LIN {X 0,Y 252.245,Z 652.898,A -85,B 0,C 180,E1 -20197.805,E2 -20197.805} C_VEL
LIN {X 0,Y 252.459,Z 653.235,A -85,B 0,C 180,E1 -20199.813,E2 -20199.813} C_VEL
LIN {X 0,Y 253.031,Z 654.37,A -85,B 0,C 180,E1 -20201.806,E2 -20201.806} C_VEL
LIN {X 0,Y 253.295,Z 655.446,A -85,B 0,C 180,E1 -20202.736,E2 -20202.736} C_VEL
LIN {X 0,Y 253.577,Z 657.958,A -85,B 0,C 180,E1 -20203.951,E2 -20203.951} C_VEL
LIN {X 0,Y 253.573,Z 661.43,A -85,B 0,C 180,E1 -20205.049,E2 -20205.049} C_VEL
LIN {X 0,Y 252.747,Z 675.435,A -85,B 0,C 180,E1 -20208.376,E2 -20208.376} C_VEL
LIN {X 0,Y 252.668,Z 684.161,A -85,B 0,C 180,E1 -20210.606,E2 -20210.606} C_VEL
LIN {X 0,Y 251.966,Z 693.895,A -85,B 0,C 180,E1 -20212.79,E2 -20212.79} C_VEL
LIN {X 0,Y 250.461,Z 703.468,A -85,B 0,C 180,E1 -20214.772,E2 -20214.772} C_VEL
LIN {X 0,Y 248.645,Z 710.196,A -85,B 0,C 180,E1 -20216.076,E2 -20216.076} C_VEL
LIN {X 0,Y 244.167,Z 721.841,A -85,B 0,C 180,E1 -20218.314,E2 -20218.314} C_VEL
LIN {X 0,Y 239.831,Z 731.637,A -85,B 0,C 180,E1 -20220.606,E2 -20220.606} C_VEL
LIN {X 0,Y 234.519,Z 741.386,A -85,B 0,C 180,E1 -20223.289,E2 -20223.289} C_VEL
LIN {X 0,Y 230.644,Z 748.224,A -85,B 0,C 180,E1 -20225.712,E2 -20225.712} C_VEL
LIN {X 0,Y 227.208,Z 753.924,A -85,B 0,C 180,E1 -20228.213,E2 -20228.213} C_VEL
LIN {X 0,Y 223.826,Z 759.888,A -85,B 0,C 180,E1 -20231.702,E2 -20231.702} C_VEL
LIN {X 0,Y 221.088,Z 764.261,A -85,B 0,C 180,E1 -20235.269,E2 -20235.269} C_VEL
LIN {X 0,Y 219.589,Z 767.051,A -85,B 0,C 180,E1 -20238.93,E2 -20238.93} C_VEL
LIN {X 0,Y 218.873,Z 768.38,A -85,B 0,C 180,E1 -20242.622,E2 -20242.622} C_VEL
LIN {X 0,Y 218.849,Z 768.456,A -85,B 0,C 180,E1 -20244.579,E2 -20244.579} C_VEL
LIN {X 0,Y 218.925,Z 768.145,A -85,B 0,C 180,E1 -20246.321,E2 -20246.321} C_VEL
LIN {X 0,Y 219.414,Z 766.339,A -85,B 0,C 180,E1 -20250.002,E2 -20250.002} C_VEL
LIN {X 0,Y 219.108,Z 763.745,A -85,B 0,C 180,E1 -20252.759,E2 -20252.759} C_VEL
LIN {X 0,Y 219.216,Z 760.085,A -85,B 0,C 180,E1 -20255.521,E2 -20255.521} C_VEL
LIN {X 0,Y 219.319,Z 755.208,A -85,B 0,C 180,E1 -20258.293,E2 -20258.293} C_VEL
LIN {X 0,Y 219.698,Z 748.98,A -85,B 0,C 180,E1 -20261.067,E2 -20261.067} C_VEL
LIN {X 0,Y 220.582,Z 741.209,A -85,B 0,C 180,E1 -20263.827,E2 -20263.827} C_VEL
LIN {X 0,Y 221.768,Z 731.543,A -85,B 0,C 180,E1 -20266.573,E2 -20266.573} C_VEL
LIN {X 0,Y 223.305,Z 720.643,A -85,B 0,C 180,E1 -20269.027,E2 -20269.027} C_VEL
LIN {X 0,Y 224.735,Z 710.679,A -85,B 0,C 180,E1 -20270.839,E2 -20270.839} C_VEL
LIN {X 0,Y 224.755,Z 697.58,A -85,B 0,C 180,E1 -20272.767,E2 -20272.767} C_VEL
LIN {X 0,Y 224.665,Z 688.245,A -85,B 0,C 180,E1 -20273.997,E2 -20273.997} C_VEL
LIN {X 0,Y 224.567,Z 676.067,A -85,B 0,C 180,E1 -20275.81,E2 -20275.81} C_VEL
LIN {X 0,Y 224.016,Z 662.677,A -85,B 0,C 180,E1 -20277.401,E2 -20277.401} C_VEL
LIN {X 0,Y 222.878,Z 649.109,A -85,B 0,C 180,E1 -20278.629,E2 -20278.629} C_VEL
LIN {X 0,Y 221.828,Z 640.058,A -85,B 0,C 180,E1 -20279.284,E2 -20279.284} C_VEL
LIN {X 0,Y 221.802,Z 634.375,A -85,B 0,C 180,E1 -20280.398,E2 -20280.398} C_VEL
LIN {X 0,Y 223.684,Z 624.514,A -85,B 0,C 180,E1 -20285.785,E2 -20285.785} C_VEL
LIN {X 0,Y 224.829,Z 619.234,A -85,B 0,C 180,E1 -20288.697,E2 -20288.697} C_VEL
LIN {X 0,Y 224.391,Z 614.928,A -85,B 0,C 180,E1 -20291.262,E2 -20291.262} C_VEL
LIN {X 0,Y 222.825,Z 607.241,A -85,B 0,C 180,E1 -20296.06,E2 -20296.06} C_VEL
LIN {X 0,Y 221.557,Z 600.491,A -85,B 0,C 180,E1 -20300.622,E2 -20300.622} C_VEL
LIN {X 0,Y 220.894,Z 596.978,A -85,B 0,C 180,E1 -20303.234,E2 -20303.234} C_VEL
LIN {X 0,Y 220.831,Z 596.982,A -85,B 0,C 180,E1 -20307.245,E2 -20307.245} C_VEL
LIN {X 0,Y 220.842,Z 596.976,A -85,B 0,C 180,E1 -20311.486,E2 -20311.486} C_VEL
LIN {X 0,Y 220.874,Z 596.971,A -85,B 0,C 180,E1 -20315.565,E2 -20315.565} C_VEL
LIN {X 0,Y 220.899,Z 596.97,A -85,B 0,C 180,E1 -20319.514,E2 -20319.514} C_VEL
LIN {X 0,Y 221.023,Z 596.954,A -85,B 0,C 180,E1 -20323.37,E2 -20323.37} C_VEL
LIN {X 0,Y 221.123,Z 596.942,A -85,B 0,C 180,E1 -20329.006,E2 -20329.006} C_VEL
LIN {X 0,Y 221.317,Z 596.917,A -85,B 0,C 180,E1 -20332.702,E2 -20332.702} C_VEL
LIN {X 0,Y 221.517,Z 596.891,A -85,B 0,C 180,E1 -20338.181,E2 -20338.181} C_VEL
LIN {X 0,Y 221.517,Z 596.888,A -85,B 0,C 180,E1 -20341.817,E2 -20341.817} C_VEL
LIN {X 0,Y 221.295,Z 596.913,A -85,B 0,C 180,E1 -20347.297,E2 -20347.297} C_VEL
LIN {X 0,Y 221.117,Z 596.94,A -85,B 0,C 180,E1 -20350.993,E2 -20350.993} C_VEL
LIN {X 0,Y 221.021,Z 596.94,A -85,B 0,C 180,E1 -20356.629,E2 -20356.629} C_VEL
LIN {X 0,Y 220.897,Z 596.97,A -85,B 0,C 180,E1 -20360.485,E2 -20360.485} C_VEL
LIN {X 0,Y 220.871,Z 596.966,A -85,B 0,C 180,E1 -20364.434,E2 -20364.434} C_VEL
LIN {X 0,Y 220.84,Z 596.969,A -85,B 0,C 180,E1 -20368.512,E2 -20368.512} C_VEL
LIN {X 0,Y 220.821,Z 596.977,A -85,B 0,C 180,E1 -20372.755,E2 -20372.755} C_VEL
LIN {X 0,Y 220.813,Z 596.977,A -85,B 0,C 180,E1 -20377.277,E2 -20377.277} C_VEL
LIN {X 0,Y 220.773,Z 596.983,A -85,B 0,C 180,E1 -20381.951,E2 -20381.951} C_VEL
LIN {X 0,Y 220.834,Z 596.974,A -85,B 0,C 180,E1 -20387.051,E2 -20387.051} C_VEL
LIN {X 0,Y 220.813,Z 596.976,A -85,B 0,C 180,E1 -20390.463,E2 -20390.463} C_VEL
LIN {X 0,Y 220.833,Z 596.97,A -85,B 0,C 180,E1 -20392.793,E2 -20392.793} C_VEL
LIN {X 0,Y 220.824,Z 596.973,A -85,B 0,C 180,E1 -20397.244,E2 -20397.244} C_VEL
LIN {X 0,Y 220.828,Z 596.977,A -85,B 0,C 180,E1 -20401.484,E2 -20401.484} C_VEL
LIN {X 0,Y 220.868,Z 596.972,A -85,B 0,C 180,E1 -20405.564,E2 -20405.564} C_VEL
LIN {X 0,Y 220.893,Z 596.969,A -85,B 0,C 180,E1 -20409.512,E2 -20409.512} C_VEL
LIN {X 0,Y 221.017,Z 596.951,A -85,B 0,C 180,E1 -20413.369,E2 -20413.369} C_VEL
LIN {X 0,Y 221.028,Z 596.951,A -85,B 0,C 180,E1 -20416.038,E2 -20416.038} C_VEL
LIN {X 0,Y 223.588,Z 603.871,A -85,B 0,C 180,E1 -20417.009,E2 -20417.009} C_VEL
LIN {X 0,Y 227.422,Z 614.702,A -85,B 0,C 180,E1 -20418.752,E2 -20418.752} C_VEL
LIN {X 0,Y 229.953,Z 624.228,A -85,B 0,C 180,E1 -20420.457,E2 -20420.457} C_VEL
LIN {X 0,Y 230.705,Z 628.301,A -85,B 0,C 180,E1 -20421.237,E2 -20421.237} C_VEL
LIN {X 0,Y 229.152,Z 638.765,A -85,B 0,C 180,E1 -20423.173,E2 -20423.173} C_VEL
LIN {X 0,Y 227.315,Z 649.11,A -85,B 0,C 180,E1 -20425.565,E2 -20425.565} C_VEL
LIN {X 0,Y 225.619,Z 658.089,A -85,B 0,C 180,E1 -20428.213,E2 -20428.213} C_VEL
LIN {X 0,Y 224.289,Z 665.333,A -85,B 0,C 180,E1 -20430.896,E2 -20430.896} C_VEL
LIN {X 0,Y 223.107,Z 671.185,A -85,B 0,C 180,E1 -20433.61,E2 -20433.61} C_VEL
LIN {X 0,Y 222.214,Z 675.812,A -85,B 0,C 180,E1 -20436.354,E2 -20436.354} C_VEL
LIN {X 0,Y 221.701,Z 679.343,A -85,B 0,C 180,E1 -20439.118,E2 -20439.118} C_VEL
LIN {X 0,Y 221.511,Z 681.12,A -85,B 0,C 180,E1 -20440.972,E2 -20440.972} C_VEL
LIN {X 0,Y 221.471,Z 682.492,A -85,B 0,C 180,E1 -20442.833,E2 -20442.833} C_VEL
LIN {X 0,Y 221.569,Z 683.473,A -85,B 0,C 180,E1 -20444.698,E2 -20444.698} C_VEL
LIN {X 0,Y 221.831,Z 684.017,A -85,B 0,C 180,E1 -20446.565,E2 -20446.565} C_VEL
LIN {X 0,Y 222.29,Z 684.143,A -85,B 0,C 180,E1 -20448.473,E2 -20448.473} C_VEL
LIN {X 0,Y 222.808,Z 683.893,A -85,B 0,C 180,E1 -20450.3,E2 -20450.3} C_VEL
LIN {X 0,Y 223.531,Z 683.233,A -85,B 0,C 180,E1 -20452.164,E2 -20452.164} C_VEL
LIN {X 0,Y 225.071,Z 681.267,A -85,B 0,C 180,E1 -20455.105,E2 -20455.105} C_VEL
LIN {X 0,Y 227.381,Z 677.38,A -85,B 0,C 180,E1 -20458.623,E2 -20458.623} C_VEL
LIN {X 0,Y 229.647,Z 673.053,A -85,B 0,C 180,E1 -20461.348,E2 -20461.348} C_VEL
LIN {X 0,Y 232.269,Z 667.442,A -85,B 0,C 180,E1 -20464.038,E2 -20464.038} C_VEL
LIN {X 0,Y 235.317,Z 660.246,A -85,B 0,C 180,E1 -20466.676,E2 -20466.676} C_VEL
LIN {X 0,Y 238.089,Z 652.814,A -85,B 0,C 180,E1 -20468.846,E2 -20468.846} C_VEL
LIN {X 0,Y 239.795,Z 647.581,A -85,B 0,C 180,E1 -20470.147,E2 -20470.147} C_VEL
LIN {X 0,Y 236.234,Z 643.736,A -85,B 0,C 180,E1 -20471.949,E2 -20471.949} C_VEL
LIN {X 0,Y 229.224,Z 637.173,A -85,B 0,C 180,E1 -20475.157,E2 -20475.157} C_VEL
LIN {X 0,Y 223.707,Z 632.758,A -85,B 0,C 180,E1 -20477.512,E2 -20477.512} C_VEL
LIN {X 0,Y 222.648,Z 630.989,A -85,B 0,C 180,E1 -20478.179,E2 -20478.179} C_VEL
LIN {X 0,Y 222.276,Z 635.847,A -85,B 0,C 180,E1 -20480.776,E2 -20480.776} C_VEL
LIN {X 0,Y 224.52,Z 650.074,A -85,B 0,C 180,E1 -20481.923,E2 -20481.923} C_VEL
LIN {X 0,Y 226.528,Z 663.63,A -85,B 0,C 180,E1 -20483.379,E2 -20483.379} C_VEL
LIN {X 0,Y 227.354,Z 670.894,A -85,B 0,C 180,E1 -20484.306,E2 -20484.306} C_VEL
LIN {X 0,Y 225.67,Z 684.053,A -85,B 0,C 180,E1 -20486.175,E2 -20486.175} C_VEL
LIN {X 0,Y 224.013,Z 695.748,A -85,B 0,C 180,E1 -20488.299,E2 -20488.299} C_VEL
LIN {X 0,Y 222.521,Z 706.372,A -85,B 0,C 180,E1 -20490.69,E2 -20490.69} C_VEL
LIN {X 0,Y 221,Z 716.568,A -85,B 0,C 180,E1 -20493.564,E2 -20493.564} C_VEL
LIN {X 0,Y 220.17,Z 723.542,A -85,B 0,C 180,E1 -20495.985,E2 -20495.985} C_VEL
LIN {X 0,Y 219.407,Z 730.071,A -85,B 0,C 180,E1 -20498.772,E2 -20498.772} C_VEL
LIN {X 0,Y 218.933,Z 734.814,A -85,B 0,C 180,E1 -20501.277,E2 -20501.277} C_VEL
LIN {X 0,Y 218.61,Z 739.736,A -85,B 0,C 180,E1 -20504.67,E2 -20504.67} C_VEL
LIN {X 0,Y 218.605,Z 742.265,A -85,B 0,C 180,E1 -20506.995,E2 -20506.995} C_VEL
LIN {X 0,Y 219.038,Z 744.947,A -85,B 0,C 180,E1 -20510.769,E2 -20510.769} C_VEL
LIN {X 0,Y 219.579,Z 745.711,A -85,B 0,C 180,E1 -20512.824,E2 -20512.824} C_VEL
LIN {X 0,Y 220.776,Z 745.89,A -85,B 0,C 180,E1 -20516.35,E2 -20516.35} C_VEL
LIN {X 0,Y 222.836,Z 744.583,A -85,B 0,C 180,E1 -20520.001,E2 -20520.001} C_VEL
LIN {X 0,Y 225.68,Z 741.694,A -85,B 0,C 180,E1 -20523.572,E2 -20523.572} C_VEL
LIN {X 0,Y 228.348,Z 738.462,A -85,B 0,C 180,E1 -20526.185,E2 -20526.185} C_VEL
LIN {X 0,Y 231.512,Z 734.232,A -85,B 0,C 180,E1 -20528.731,E2 -20528.731} C_VEL
LIN {X 0,Y 235.767,Z 727.99,A -85,B 0,C 180,E1 -20531.608,E2 -20531.608} C_VEL
LIN {X 0,Y 240.003,Z 721.133,A -85,B 0,C 180,E1 -20534.004,E2 -20534.004} C_VEL
LIN {X 0,Y 244.573,Z 713.037,A -85,B 0,C 180,E1 -20536.271,E2 -20536.271} C_VEL
LIN {X 0,Y 249.602,Z 703.046,A -85,B 0,C 180,E1 -20538.468,E2 -20538.468} C_VEL
LIN {X 0,Y 252.241,Z 697.161,A -85,B 0,C 180,E1 -20539.533,E2 -20539.533} C_VEL
LIN {X 0,Y 252.802,Z 694.541,A -85,B 0,C 180,E1 -20540.201,E2 -20540.201} C_VEL
LIN {X 0,Y 253.313,Z 686.369,A -85,B 0,C 180,E1 -20542.556,E2 -20542.556} C_VEL
LIN {X 0,Y 253.154,Z 677.893,A -85,B 0,C 180,E1 -20545.251,E2 -20545.251} C_VEL
LIN {X 0,Y 252.633,Z 670.904,A -85,B 0,C 180,E1 -20547.784,E2 -20547.784} C_VEL
LIN {X 0,Y 252.207,Z 668.05,A -85,B 0,C 180,E1 -20549.092,E2 -20549.092} C_VEL
LIN {X 0,Y 251.002,Z 663.368,A -85,B 0,C 180,E1 -20552.141,E2 -20552.141} C_VEL
LIN {X 0,Y 250.022,Z 660.392,A -85,B 0,C 180,E1 -20556.179,E2 -20556.179} C_VEL
LIN {X 0,Y 250.107,Z 659.658,A -85,B 0,C 180,E1 -20558.186,E2 -20558.186} C_VEL
LIN {X 0,Y 250.545,Z 660.411,A -85,B 0,C 180,E1 -20560.77,E2 -20560.77} C_VEL
LIN {X 0,Y 250.953,Z 661.841,A -85,B 0,C 180,E1 -20562.303,E2 -20562.303} C_VEL
LIN {X 0,Y 252.479,Z 667.322,A -85,B 0,C 180,E1 -20565.904,E2 -20565.904} C_VEL
LIN {X 0,Y 252.76,Z 670.488,A -85,B 0,C 180,E1 -20567.023,E2 -20567.023} C_VEL
LIN {X 0,Y 252.747,Z 675.435,A -85,B 0,C 180,E1 -20568.376,E2 -20568.376} C_VEL
LIN {X 0,Y 252.392,Z 679.725,A -85,B 0,C 180,E1 -20569.294,E2 -20569.294} C_VEL
LIN {X 0,Y 251.368,Z 684.518,A -85,B 0,C 180,E1 -20570.061,E2 -20570.061} C_VEL
LIN {X 0,Y 247.481,Z 697.648,A -85,B 0,C 180,E1 -20571.989,E2 -20571.989} C_VEL
LIN {X 0,Y 246.749,Z 700.631,A -85,B 0,C 180,E1 -20572.586,E2 -20572.586} C_VEL
LIN {X 0,Y 244.622,Z 709.219,A -85,B 0,C 180,E1 -20574.429,E2 -20574.429} C_VEL
LIN {X 0,Y 241.616,Z 717.039,A -85,B 0,C 180,E1 -20575.951,E2 -20575.951} C_VEL
LIN {X 0,Y 236.854,Z 727.366,A -85,B 0,C 180,E1 -20578.221,E2 -20578.221} C_VEL
LIN {X 0,Y 232.207,Z 736.247,A -85,B 0,C 180,E1 -20580.542,E2 -20580.542} C_VEL
LIN {X 0,Y 226.841,Z 744.931,A -85,B 0,C 180,E1 -20583.307,E2 -20583.307} C_VEL
LIN {X 0,Y 223.111,Z 751.056,A -85,B 0,C 180,E1 -20585.829,E2 -20585.829} C_VEL
LIN {X 0,Y 219.44,Z 756.501,A -85,B 0,C 180,E1 -20588.648,E2 -20588.648} C_VEL
LIN {X 0,Y 216.301,Z 761.358,A -85,B 0,C 180,E1 -20592.023,E2 -20592.023} C_VEL
LIN {X 0,Y 214.218,Z 764.263,A -85,B 0,C 180,E1 -20594.786,E2 -20594.786} C_VEL
LIN {X 0,Y 212.574,Z 766.842,A -85,B 0,C 180,E1 -20598.56,E2 -20598.56} C_VEL
LIN {X 0,Y 212.1,Z 767.581,A -85,B 0,C 180,E1 -20600.465,E2 -20600.465} C_VEL
LIN {X 0,Y 211.772,Z 767.892,A -85,B 0,C 180,E1 -20604.288,E2 -20604.288} C_VEL
LIN {X 0,Y 211.859,Z 767.493,A -85,B 0,C 180,E1 -20606.198,E2 -20606.198} C_VEL
LIN {X 0,Y 211.921,Z 766.687,A -85,B 0,C 180,E1 -20608.101,E2 -20608.101} C_VEL
LIN {X 0,Y 212.356,Z 765.482,A -85,B 0,C 180,E1 -20610.002,E2 -20610.002} C_VEL
LIN {X 0,Y 212.086,Z 762.722,A -85,B 0,C 180,E1 -20612.851,E2 -20612.851} C_VEL
LIN {X 0,Y 212.159,Z 758.892,A -85,B 0,C 180,E1 -20615.705,E2 -20615.705} C_VEL
LIN {X 0,Y 212.293,Z 753.825,A -85,B 0,C 180,E1 -20618.569,E2 -20618.569} C_VEL
LIN {X 0,Y 212.73,Z 747.381,A -85,B 0,C 180,E1 -20621.435,E2 -20621.435} C_VEL
LIN {X 0,Y 213.635,Z 739.368,A -85,B 0,C 180,E1 -20624.286,E2 -20624.286} C_VEL
LIN {X 0,Y 214.686,Z 731.164,A -85,B 0,C 180,E1 -20626.647,E2 -20626.647} C_VEL
LIN {X 0,Y 216.273,Z 720.163,A -85,B 0,C 180,E1 -20629.205,E2 -20629.205} C_VEL
LIN {X 0,Y 217.672,Z 710.332,A -85,B 0,C 180,E1 -20631.052,E2 -20631.052} C_VEL
LIN {X 0,Y 217.723,Z 699.102,A -85,B 0,C 180,E1 -20632.792,E2 -20632.792} C_VEL
LIN {X 0,Y 217.669,Z 691.704,A -85,B 0,C 180,E1 -20633.805,E2 -20633.805} C_VEL
LIN {X 0,Y 217.728,Z 680.37,A -85,B 0,C 180,E1 -20635.717,E2 -20635.717} C_VEL
LIN {X 0,Y 217.496,Z 667.855,A -85,B 0,C 180,E1 -20637.42,E2 -20637.42} C_VEL
LIN {X 0,Y 216.673,Z 654.932,A -85,B 0,C 180,E1 -20638.808,E2 -20638.808} C_VEL
LIN {X 0,Y 215.186,Z 640.623,A -85,B 0,C 180,E1 -20639.963,E2 -20639.963} C_VEL
LIN {X 0,Y 214.937,Z 638.555,A -85,B 0,C 180,E1 -20640.115,E2 -20640.115} C_VEL
LIN {X 0,Y 214.908,Z 633.563,A -85,B 0,C 180,E1 -20641.14,E2 -20641.14} C_VEL
LIN {X 0,Y 216.56,Z 625.373,A -85,B 0,C 180,E1 -20645.774,E2 -20645.774} C_VEL
LIN {X 0,Y 217.809,Z 619.336,A -85,B 0,C 180,E1 -20649.248,E2 -20649.248} C_VEL
LIN {X 0,Y 217.189,Z 614.995,A -85,B 0,C 180,E1 -20651.904,E2 -20651.904} C_VEL
LIN {X 0,Y 215.661,Z 607.527,A -85,B 0,C 180,E1 -20656.814,E2 -20656.814} C_VEL
LIN {X 0,Y 214.308,Z 600.328,A -85,B 0,C 180,E1 -20661.913,E2 -20661.913} C_VEL
LIN {X 0,Y 213.843,Z 597.857,A -85,B 0,C 180,E1 -20663.839,E2 -20663.839} C_VEL
LIN {X 0,Y 213.802,Z 597.856,A -85,B 0,C 180,E1 -20668.724,E2 -20668.724} C_VEL
LIN {X 0,Y 213.832,Z 597.849,A -85,B 0,C 180,E1 -20672.603,E2 -20672.603} C_VEL
LIN {X 0,Y 213.859,Z 597.845,A -85,B 0,C 180,E1 -20676.953,E2 -20676.953} C_VEL
LIN {X 0,Y 213.95,Z 597.836,A -85,B 0,C 180,E1 -20682.803,E2 -20682.803} C_VEL
LIN {X 0,Y 213.987,Z 597.831,A -85,B 0,C 180,E1 -20686.708,E2 -20686.708} C_VEL
LIN {X 0,Y 214.203,Z 597.804,A -85,B 0,C 180,E1 -20690.557,E2 -20690.557} C_VEL
LIN {X 0,Y 214.254,Z 597.797,A -85,B 0,C 180,E1 -20692.46,E2 -20692.46} C_VEL
LIN {X 0,Y 214.451,Z 597.771,A -85,B 0,C 180,E1 -20698.121,E2 -20698.121} C_VEL
LIN {X 0,Y 214.556,Z 597.759,A -85,B 0,C 180,E1 -20699.999,E2 -20699.999} C_VEL
LIN {X 0,Y 214.45,Z 597.768,A -85,B 0,C 180,E1 -20701.877,E2 -20701.877} C_VEL
LIN {X 0,Y 214.233,Z 597.792,A -85,B 0,C 180,E1 -20707.539,E2 -20707.539} C_VEL
LIN {X 0,Y 214.049,Z 597.82,A -85,B 0,C 180,E1 -20711.361,E2 -20711.361} C_VEL
LIN {X 0,Y 213.936,Z 597.82,A -85,B 0,C 180,E1 -20715.236,E2 -20715.236} C_VEL
LIN {X 0,Y 213.844,Z 597.844,A -85,B 0,C 180,E1 -20719.186,E2 -20719.186} C_VEL
LIN {X 0,Y 213.852,Z 597.843,A -85,B 0,C 180,E1 -20723.226,E2 -20723.226} C_VEL
LIN {X 0,Y 213.833,Z 597.836,A -85,B 0,C 180,E1 -20727.448,E2 -20727.448} C_VEL
LIN {X 0,Y 213.78,Z 597.854,A -85,B 0,C 180,E1 -20731.735,E2 -20731.735} C_VEL
LIN {X 0,Y 213.747,Z 597.86,A -85,B 0,C 180,E1 -20736.287,E2 -20736.287} C_VEL
LIN {X 0,Y 213.715,Z 597.862,A -85,B 0,C 180,E1 -20741.124,E2 -20741.124} C_VEL
LIN {X 0,Y 213.779,Z 597.847,A -85,B 0,C 180,E1 -20746.338,E2 -20746.338} C_VEL
LIN {X 0,Y 213.739,Z 597.852,A -85,B 0,C 180,E1 -20751.335,E2 -20751.335} C_VEL
LIN {X 0,Y 213.771,Z 597.856,A -85,B 0,C 180,E1 -20756.019,E2 -20756.019} C_VEL
LIN {X 0,Y 213.761,Z 597.859,A -85,B 0,C 180,E1 -20760.449,E2 -20760.449} C_VEL
LIN {X 0,Y 213.802,Z 597.853,A -85,B 0,C 180,E1 -20764.7,E2 -20764.7} C_VEL
LIN {X 0,Y 213.814,Z 597.853,A -85,B 0,C 180,E1 -20768.802,E2 -20768.802} C_VEL
LIN {X 0,Y 213.944,Z 597.834,A -85,B 0,C 180,E1 -20772.802,E2 -20772.802} C_VEL
LIN {X 0,Y 213.967,Z 597.91,A -85,B 0,C 180,E1 -20775.233,E2 -20775.233} C_VEL
LIN {X 0,Y 217.501,Z 607.238,A -85,B 0,C 180,E1 -20776.639,E2 -20776.639} C_VEL
LIN {X 0,Y 220.812,Z 616.808,A -85,B 0,C 180,E1 -20778.277,E2 -20778.277} C_VEL
LIN {X 0,Y 223.197,Z 625.637,A -85,B 0,C 180,E1 -20779.944,E2 -20779.944} C_VEL
LIN {X 0,Y 223.95,Z 629.806,A -85,B 0,C 180,E1 -20780.778,E2 -20780.778} C_VEL
LIN {X 0,Y 222.375,Z 640.022,A -85,B 0,C 180,E1 -20782.736,E2 -20782.736} C_VEL
LIN {X 0,Y 220.611,Z 649.483,A -85,B 0,C 180,E1 -20784.972,E2 -20784.972} C_VEL
LIN {X 0,Y 218.837,Z 658.584,A -85,B 0,C 180,E1 -20787.698,E2 -20787.698} C_VEL
LIN {X 0,Y 217.404,Z 665.924,A -85,B 0,C 180,E1 -20790.461,E2 -20790.461} C_VEL
LIN {X 0,Y 215.974,Z 672.721,A -85,B 0,C 180,E1 -20793.73,E2 -20793.73} C_VEL
LIN {X 0,Y 215.119,Z 677.223,A -85,B 0,C 180,E1 -20796.564,E2 -20796.564} C_VEL
LIN {X 0,Y 214.618,Z 680.651,A -85,B 0,C 180,E1 -20799.422,E2 -20799.422} C_VEL
LIN {X 0,Y 214.453,Z 682.376,A -85,B 0,C 180,E1 -20801.338,E2 -20801.338} C_VEL
LIN {X 0,Y 214.441,Z 683.7,A -85,B 0,C 180,E1 -20803.261,E2 -20803.261} C_VEL
LIN {X 0,Y 214.607,Z 684.601,A -85,B 0,C 180,E1 -20805.186,E2 -20805.186} C_VEL
LIN {X 0,Y 215.394,Z 685.157,A -85,B 0,C 180,E1 -20809.042,E2 -20809.042} C_VEL
LIN {X 0,Y 216.007,Z 684.855,A -85,B 0,C 180,E1 -20810.969,E2 -20810.969} C_VEL
LIN {X 0,Y 216.821,Z 684.095,A -85,B 0,C 180,E1 -20812.888,E2 -20812.888} C_VEL
LIN {X 0,Y 218.344,Z 682.239,A -85,B 0,C 180,E1 -20815.678,E2 -20815.678} C_VEL
LIN {X 0,Y 220.274,Z 679.241,A -85,B 0,C 180,E1 -20818.591,E2 -20818.591} C_VEL
LIN {X 0,Y 222.725,Z 674.878,A -85,B 0,C 180,E1 -20821.575,E2 -20821.575} C_VEL
LIN {X 0,Y 225.717,Z 668.854,A -85,B 0,C 180,E1 -20824.625,E2 -20824.625} C_VEL
LIN {X 0,Y 228.61,Z 662.508,A -85,B 0,C 180,E1 -20827.084,E2 -20827.084} C_VEL
LIN {X 0,Y 231.812,Z 654.469,A -85,B 0,C 180,E1 -20829.541,E2 -20829.541} C_VEL
LIN {X 0,Y 233.082,Z 651.055,A -85,B 0,C 180,E1 -20830.428,E2 -20830.428} C_VEL
LIN {X 0,Y 232.462,Z 649.941,A -85,B 0,C 180,E1 -20830.904,E2 -20830.904} C_VEL
LIN {X 0,Y 227.146,Z 644.905,A -85,B 0,C 180,E1 -20833.587,E2 -20833.587} C_VEL
LIN {X 0,Y 222.301,Z 640.532,A -85,B 0,C 180,E1 -20835.932,E2 -20835.932} C_VEL
LIN {X 0,Y 216.034,Z 635.517,A -85,B 0,C 180,E1 -20838.857,E2 -20838.857} C_VEL
LIN {X 0,Y 215.428,Z 634.282,A -85,B 0,C 180,E1 -20839.354,E2 -20839.354} C_VEL
LIN {X 0,Y 215.285,Z 635.964,A -85,B 0,C 180,E1 -20840.29,E2 -20840.29} C_VEL
LIN {X 0,Y 217.629,Z 651.221,A -85,B 0,C 180,E1 -20841.617,E2 -20841.617} C_VEL
LIN {X 0,Y 219.581,Z 664.784,A -85,B 0,C 180,E1 -20843.142,E2 -20843.142} C_VEL
LIN {X 0,Y 220.374,Z 670.376,A -85,B 0,C 180,E1 -20843.887,E2 -20843.887} C_VEL
LIN {X 0,Y 218.947,Z 682,A -85,B 0,C 180,E1 -20845.547,E2 -20845.547} C_VEL
LIN {X 0,Y 217.416,Z 693.05,A -85,B 0,C 180,E1 -20847.5,E2 -20847.5} C_VEL
LIN {X 0,Y 215.939,Z 703.184,A -85,B 0,C 180,E1 -20849.705,E2 -20849.705} C_VEL
LIN {X 0,Y 214.51,Z 712.508,A -85,B 0,C 180,E1 -20852.198,E2 -20852.198} C_VEL
LIN {X 0,Y 213.33,Z 721.502,A -85,B 0,C 180,E1 -20855.164,E2 -20855.164} C_VEL
LIN {X 0,Y 212.527,Z 727.963,A -85,B 0,C 180,E1 -20857.802,E2 -20857.802} C_VEL
LIN {X 0,Y 211.939,Z 733.605,A -85,B 0,C 180,E1 -20860.635,E2 -20860.635} C_VEL
LIN {X 0,Y 211.582,Z 738.416,A -85,B 0,C 180,E1 -20863.7,E2 -20863.7} C_VEL
LIN {X 0,Y 211.485,Z 741.802,A -85,B 0,C 180,E1 -20866.549,E2 -20866.549} C_VEL
LIN {X 0,Y 211.589,Z 743.577,A -85,B 0,C 180,E1 -20868.505,E2 -20868.505} C_VEL
LIN {X 0,Y 211.865,Z 744.921,A -85,B 0,C 180,E1 -20870.454,E2 -20870.454} C_VEL
LIN {X 0,Y 212.485,Z 745.993,A -85,B 0,C 180,E1 -20872.848,E2 -20872.848} C_VEL
LIN {X 0,Y 213.626,Z 746.508,A -85,B 0,C 180,E1 -20876.228,E2 -20876.228} C_VEL
LIN {X 0,Y 215.704,Z 745.599,A -85,B 0,C 180,E1 -20880.001,E2 -20880.001} C_VEL
LIN {X 0,Y 218.617,Z 743.182,A -85,B 0,C 180,E1 -20883.687,E2 -20883.687} C_VEL
LIN {X 0,Y 221.321,Z 740.321,A -85,B 0,C 180,E1 -20886.382,E2 -20886.382} C_VEL
LIN {X 0,Y 224.599,Z 736.503,A -85,B 0,C 180,E1 -20889.002,E2 -20889.002} C_VEL
LIN {X 0,Y 228.331,Z 731.634,A -85,B 0,C 180,E1 -20891.542,E2 -20891.542} C_VEL
LIN {X 0,Y 233.263,Z 724.547,A -85,B 0,C 180,E1 -20894.393,E2 -20894.393} C_VEL
LIN {X 0,Y 238.055,Z 716.965,A -85,B 0,C 180,E1 -20896.73,E2 -20896.73} C_VEL
LIN {X 0,Y 243.241,Z 707.803,A -85,B 0,C 180,E1 -20898.969,E2 -20898.969} C_VEL
LIN {X 0,Y 246.905,Z 700.594,A -85,B 0,C 180,E1 -20900.408,E2 -20900.408} C_VEL
LIN {X 0,Y 247.607,Z 698.809,A -85,B 0,C 180,E1 -20900.782,E2 -20900.782} C_VEL
LIN {X 0,Y 248.563,Z 691.931,A -85,B 0,C 180,E1 -20902.881,E2 -20902.881} C_VEL
LIN {X 0,Y 249,Z 683.501,A -85,B 0,C 180,E1 -20905.703,E2 -20905.703} C_VEL
LIN {X 0,Y 249.005,Z 676.875,A -85,B 0,C 180,E1 -20908.189,E2 -20908.189} C_VEL
LIN {X 0,Y 248.766,Z 673.67,A -85,B 0,C 180,E1 -20909.728,E2 -20909.728} C_VEL
LIN {X 0,Y 248.039,Z 669.604,A -85,B 0,C 180,E1 -20912.572,E2 -20912.572} C_VEL
LIN {X 0,Y 247.521,Z 666.878,A -85,B 0,C 180,E1 -20916.604,E2 -20916.604} C_VEL
LIN {X 0,Y 247.698,Z 666.446,A -85,B 0,C 180,E1 -20918.625,E2 -20918.625} C_VEL
LIN {X 0,Y 248.047,Z 667.091,A -85,B 0,C 180,E1 -20920.668,E2 -20920.668} C_VEL
LIN {X 0,Y 248.449,Z 669.351,A -85,B 0,C 180,E1 -20922.759,E2 -20922.759} C_VEL
LIN {X 0,Y 249.286,Z 672.962,A -85,B 0,C 180,E1 -20925.188,E2 -20925.188} C_VEL
LIN {X 0,Y 249.373,Z 675.951,A -85,B 0,C 180,E1 -20926.295,E2 -20926.295} C_VEL
LIN {X 0,Y 248.73,Z 686.204,A -85,B 0,C 180,E1 -20929.164,E2 -20929.164} C_VEL
LIN {X 0,Y 247.447,Z 696.646,A -85,B 0,C 180,E1 -20931.684,E2 -20931.684} C_VEL
LIN {X 0,Y 246.749,Z 700.631,A -85,B 0,C 180,E1 -20932.586,E2 -20932.586} C_VEL
LIN {X 0,Y 245.893,Z 703.651,A -85,B 0,C 180,E1 -20933.161,E2 -20933.161} C_VEL
LIN {X 0,Y 244.553,Z 706.757,A -85,B 0,C 180,E1 -20933.634,E2 -20933.634} C_VEL
LIN {X 0,Y 240.956,Z 713.132,A -85,B 0,C 180,E1 -20934.405,E2 -20934.405} C_VEL
LIN {X 0,Y 235.938,Z 720.792,A -85,B 0,C 180,E1 -20935.401,E2 -20935.401} C_VEL
LIN {X 0,Y 233.43,Z 725.032,A -85,B 0,C 180,E1 -20936.231,E2 -20936.231} C_VEL
LIN {X 0,Y 227.88,Z 735.142,A -85,B 0,C 180,E1 -20938.899,E2 -20938.899} C_VEL
LIN {X 0,Y 222.133,Z 743.929,A -85,B 0,C 180,E1 -20941.67,E2 -20941.67} C_VEL
LIN {X 0,Y 217.912,Z 750.069,A -85,B 0,C 180,E1 -20944.192,E2 -20944.192} C_VEL
LIN {X 0,Y 213.455,Z 756.156,A -85,B 0,C 180,E1 -20947.405,E2 -20947.405} C_VEL
LIN {X 0,Y 210.378,Z 760.482,A -85,B 0,C 180,E1 -20950.486,E2 -20950.486} C_VEL
LIN {X 0,Y 207.369,Z 764.283,A -85,B 0,C 180,E1 -20954.27,E2 -20954.27} C_VEL
LIN {X 0,Y 205.572,Z 766.581,A -85,B 0,C 180,E1 -20958.165,E2 -20958.165} C_VEL
LIN {X 0,Y 204.771,Z 767.428,A -85,B 0,C 180,E1 -20962.111,E2 -20962.111} C_VEL
LIN {X 0,Y 204.795,Z 766.806,A -85,B 0,C 180,E1 -20966.066,E2 -20966.066} C_VEL
LIN {X 0,Y 205.299,Z 764.571,A -85,B 0,C 180,E1 -20970.002,E2 -20970.002} C_VEL
LIN {X 0,Y 205.063,Z 761.632,A -85,B 0,C 180,E1 -20972.949,E2 -20972.949} C_VEL
LIN {X 0,Y 205.138,Z 757.603,A -85,B 0,C 180,E1 -20975.901,E2 -20975.901} C_VEL
LIN {X 0,Y 205.266,Z 752.318,A -85,B 0,C 180,E1 -20978.865,E2 -20978.865} C_VEL
LIN {X 0,Y 205.768,Z 745.673,A -85,B 0,C 180,E1 -20981.827,E2 -20981.827} C_VEL
LIN {X 0,Y 206.724,Z 737.351,A -85,B 0,C 180,E1 -20984.774,E2 -20984.774} C_VEL
LIN {X 0,Y 207.863,Z 728.899,A -85,B 0,C 180,E1 -20987.21,E2 -20987.21} C_VEL
LIN {X 0,Y 209.384,Z 718.669,A -85,B 0,C 180,E1 -20989.614,E2 -20989.614} C_VEL
LIN {X 0,Y 210.601,Z 709.754,A -85,B 0,C 180,E1 -20991.321,E2 -20991.321} C_VEL
LIN {X 0,Y 210.668,Z 696.957,A -85,B 0,C 180,E1 -20993.34,E2 -20993.34} C_VEL
LIN {X 0,Y 210.68,Z 693.582,A -85,B 0,C 180,E1 -20993.86,E2 -20993.86} C_VEL
LIN {X 0,Y 210.833,Z 681.813,A -85,B 0,C 180,E1 -20996.02,E2 -20996.02} C_VEL
LIN {X 0,Y 210.731,Z 669.4,A -85,B 0,C 180,E1 -20997.835,E2 -20997.835} C_VEL
LIN {X 0,Y 210.08,Z 657.008,A -85,B 0,C 180,E1 -20999.295,E2 -20999.295} C_VEL
LIN {X 0,Y 208.869,Z 643.323,A -85,B 0,C 180,E1 -21000.54,E2 -21000.54} C_VEL
LIN {X 0,Y 208.048,Z 637.114,A -85,B 0,C 180,E1 -21001.01,E2 -21001.01} C_VEL
LIN {X 0,Y 208.053,Z 632.591,A -85,B 0,C 180,E1 -21002.014,E2 -21002.014} C_VEL
LIN {X 0,Y 209.953,Z 624.026,A -85,B 0,C 180,E1 -21007.054,E2 -21007.054} C_VEL
LIN {X 0,Y 210.748,Z 620.203,A -85,B 0,C 180,E1 -21009.319,E2 -21009.319} C_VEL
LIN {X 0,Y 209.954,Z 615.147,A -85,B 0,C 180,E1 -21012.571,E2 -21012.571} C_VEL
LIN {X 0,Y 208.48,Z 607.844,A -85,B 0,C 180,E1 -21017.606,E2 -21017.606} C_VEL
LIN {X 0,Y 207.296,Z 601.32,A -85,B 0,C 180,E1 -21022.391,E2 -21022.391} C_VEL
LIN {X 0,Y 206.77,Z 598.739,A -85,B 0,C 180,E1 -21024.433,E2 -21024.433} C_VEL
LIN {X 0,Y 206.73,Z 598.736,A -85,B 0,C 180,E1 -21029.339,E2 -21029.339} C_VEL
LIN {X 0,Y 206.739,Z 598.732,A -85,B 0,C 180,E1 -21033.772,E2 -21033.772} C_VEL
LIN {X 0,Y 206.765,Z 598.73,A -85,B 0,C 180,E1 -21038.043,E2 -21038.043} C_VEL
LIN {X 0,Y 206.88,Z 598.719,A -85,B 0,C 180,E1 -21042.196,E2 -21042.196} C_VEL
LIN {X 0,Y 206.92,Z 598.715,A -85,B 0,C 180,E1 -21046.245,E2 -21046.245} C_VEL
LIN {X 0,Y 207.139,Z 598.686,A -85,B 0,C 180,E1 -21050.232,E2 -21050.232} C_VEL
LIN {X 0,Y 207.195,Z 598.675,A -85,B 0,C 180,E1 -21052.201,E2 -21052.201} C_VEL
LIN {X 0,Y 207.387,Z 598.651,A -85,B 0,C 180,E1 -21058.057,E2 -21058.057} C_VEL
LIN {X 0,Y 207.521,Z 598.635,A -85,B 0,C 180,E1 -21059.999,E2 -21059.999} C_VEL
LIN {X 0,Y 207.387,Z 598.647,A -85,B 0,C 180,E1 -21061.941,E2 -21061.941} C_VEL
LIN {X 0,Y 207.173,Z 598.672,A -85,B 0,C 180,E1 -21067.798,E2 -21067.798} C_VEL
LIN {X 0,Y 206.986,Z 598.7,A -85,B 0,C 180,E1 -21071.754,E2 -21071.754} C_VEL
LIN {X 0,Y 206.87,Z 598.699,A -85,B 0,C 180,E1 -21075.77,E2 -21075.77} C_VEL
LIN {X 0,Y 206.788,Z 598.723,A -85,B 0,C 180,E1 -21079.868,E2 -21079.868} C_VEL
LIN {X 0,Y 206.768,Z 598.725,A -85,B 0,C 180,E1 -21084.071,E2 -21084.071} C_VEL
LIN {X 0,Y 206.748,Z 598.722,A -85,B 0,C 180,E1 -21088.417,E2 -21088.417} C_VEL
LIN {X 0,Y 206.706,Z 598.734,A -85,B 0,C 180,E1 -21092.955,E2 -21092.955} C_VEL
LIN {X 0,Y 206.683,Z 598.738,A -85,B 0,C 180,E1 -21097.738,E2 -21097.738} C_VEL
LIN {X 0,Y 206.645,Z 598.742,A -85,B 0,C 180,E1 -21101.561,E2 -21101.561} C_VEL
LIN {X 0,Y 206.68,Z 598.728,A -85,B 0,C 180,E1 -21105.567,E2 -21105.567} C_VEL
LIN {X 0,Y 206.681,Z 598.737,A -85,B 0,C 180,E1 -21109.752,E2 -21109.752} C_VEL
LIN {X 0,Y 206.733,Z 598.734,A -85,B 0,C 180,E1 -21114.693,E2 -21114.693} C_VEL
LIN {X 0,Y 206.708,Z 598.734,A -85,B 0,C 180,E1 -21119.335,E2 -21119.335} C_VEL
LIN {X 0,Y 206.733,Z 598.728,A -85,B 0,C 180,E1 -21123.77,E2 -21123.77} C_VEL
LIN {X 0,Y 206.758,Z 598.728,A -85,B 0,C 180,E1 -21128.042,E2 -21128.042} C_VEL
LIN {X 0,Y 206.874,Z 598.718,A -85,B 0,C 180,E1 -21132.195,E2 -21132.195} C_VEL
LIN {X 0,Y 206.882,Z 598.706,A -85,B 0,C 180,E1 -21134.324,E2 -21134.324} C_VEL
LIN {X 0,Y 210.29,Z 607.542,A -85,B 0,C 180,E1 -21135.739,E2 -21135.739} C_VEL
LIN {X 0,Y 214.15,Z 618.59,A -85,B 0,C 180,E1 -21137.716,E2 -21137.716} C_VEL
LIN {X 0,Y 216.696,Z 628.229,A -85,B 0,C 180,E1 -21139.639,E2 -21139.639} C_VEL
LIN {X 0,Y 217.158,Z 630.75,A -85,B 0,C 180,E1 -21140.174,E2 -21140.174} C_VEL
LIN {X 0,Y 215.571,Z 641.287,A -85,B 0,C 180,E1 -21142.27,E2 -21142.27} C_VEL
LIN {X 0,Y 213.909,Z 649.823,A -85,B 0,C 180,E1 -21144.342,E2 -21144.342} C_VEL
LIN {X 0,Y 212.333,Z 657.689,A -85,B 0,C 180,E1 -21146.678,E2 -21146.678} C_VEL
LIN {X 0,Y 210.849,Z 665.053,A -85,B 0,C 180,E1 -21149.377,E2 -21149.377} C_VEL
LIN {X 0,Y 209.632,Z 670.689,A -85,B 0,C 180,E1 -21151.919,E2 -21151.919} C_VEL
LIN {X 0,Y 208.54,Z 675.849,A -85,B 0,C 180,E1 -21154.831,E2 -21154.831} C_VEL
LIN {X 0,Y 207.818,Z 679.872,A -85,B 0,C 180,E1 -21157.772,E2 -21157.772} C_VEL
LIN {X 0,Y 207.463,Z 682.888,A -85,B 0,C 180,E1 -21160.769,E2 -21160.769} C_VEL
LIN {X 0,Y 207.449,Z 684.894,A -85,B 0,C 180,E1 -21163.716,E2 -21163.716} C_VEL
LIN {X 0,Y 208.03,Z 686.13,A -85,B 0,C 180,E1 -21167.699,E2 -21167.699} C_VEL
LIN {X 0,Y 208.544,Z 686.17,A -85,B 0,C 180,E1 -21169.692,E2 -21169.692} C_VEL
LIN {X 0,Y 209.236,Z 685.782,A -85,B 0,C 180,E1 -21171.681,E2 -21171.681} C_VEL
LIN {X 0,Y 210.14,Z 684.956,A -85,B 0,C 180,E1 -21173.659,E2 -21173.659} C_VEL
LIN {X 0,Y 211.631,Z 683.217,A -85,B 0,C 180,E1 -21176.283,E2 -21176.283} C_VEL
LIN {X 0,Y 213.893,Z 679.889,A -85,B 0,C 180,E1 -21179.527,E2 -21179.527} C_VEL
LIN {X 0,Y 216.31,Z 675.797,A -85,B 0,C 180,E1 -21182.356,E2 -21182.356} C_VEL
LIN {X 0,Y 219.208,Z 670.265,A -85,B 0,C 180,E1 -21185.244,E2 -21185.244} C_VEL
LIN {X 0,Y 222.623,Z 663.091,A -85,B 0,C 180,E1 -21188.1,E2 -21188.1} C_VEL
LIN {X 0,Y 226.189,Z 654.487,A -85,B 0,C 180,E1 -21190.728,E2 -21190.728} C_VEL
LIN {X 0,Y 225.355,Z 652.709,A -85,B 0,C 180,E1 -21191.543,E2 -21191.543} C_VEL
LIN {X 0,Y 218.774,Z 646.735,A -85,B 0,C 180,E1 -21195.031,E2 -21195.031} C_VEL
LIN {X 0,Y 210.254,Z 639.917,A -85,B 0,C 180,E1 -21199.323,E2 -21199.323} C_VEL
LIN {X 0,Y 208.838,Z 639.161,A -85,B 0,C 180,E1 -21199.939,E2 -21199.939} C_VEL
LIN {X 0,Y 208.658,Z 638.98,A -85,B 0,C 180,E1 -21200.104,E2 -21200.104} C_VEL
LIN {X 0,Y 210.799,Z 653.071,A -85,B 0,C 180,E1 -21201.386,E2 -21201.386} C_VEL
LIN {X 0,Y 212.566,Z 665.305,A -85,B 0,C 180,E1 -21202.821,E2 -21202.821} C_VEL
LIN {X 0,Y 213.362,Z 671.221,A -85,B 0,C 180,E1 -21203.637,E2 -21203.637} C_VEL
LIN {X 0,Y 211.63,Z 684.377,A -85,B 0,C 180,E1 -21205.63,E2 -21205.63} C_VEL
LIN {X 0,Y 209.888,Z 696.098,A -85,B 0,C 180,E1 -21207.89,E2 -21207.89} C_VEL
LIN {X 0,Y 208.274,Z 707.033,A -85,B 0,C 180,E1 -21210.513,E2 -21210.513} C_VEL
LIN {X 0,Y 206.874,Z 716.2,A -85,B 0,C 180,E1 -21213.249,E2 -21213.249} C_VEL
LIN {X 0,Y 205.842,Z 724.469,A -85,B 0,C 180,E1 -21216.281,E2 -21216.281} C_VEL
LIN {X 0,Y 205.192,Z 730.322,A -85,B 0,C 180,E1 -21218.923,E2 -21218.923} C_VEL
LIN {X 0,Y 204.672,Z 735.813,A -85,B 0,C 180,E1 -21221.999,E2 -21221.999} C_VEL
LIN {X 0,Y 204.433,Z 740.171,A -85,B 0,C 180,E1 -21225.168,E2 -21225.168} C_VEL
LIN {X 0,Y 204.446,Z 743.204,A -85,B 0,C 180,E1 -21228.098,E2 -21228.098} C_VEL
LIN {X 0,Y 205.166,Z 745.903,A -85,B 0,C 180,E1 -21232.125,E2 -21232.125} C_VEL
LIN {X 0,Y 205.744,Z 746.658,A -85,B 0,C 180,E1 -21234.119,E2 -21234.119} C_VEL
LIN {X 0,Y 207.364,Z 746.944,A -85,B 0,C 180,E1 -21238.059,E2 -21238.059} C_VEL
LIN {X 0,Y 209.927,Z 745.737,A -85,B 0,C 180,E1 -21241.919,E2 -21241.919} C_VEL
LIN {X 0,Y 213.298,Z 742.99,A -85,B 0,C 180,E1 -21245.674,E2 -21245.674} C_VEL
LIN {X 0,Y 216.47,Z 739.877,A -85,B 0,C 180,E1 -21248.402,E2 -21248.402} C_VEL
LIN {X 0,Y 221.51,Z 734.242,A -85,B 0,C 180,E1 -21251.902,E2 -21251.902} C_VEL
LIN {X 0,Y 226.575,Z 727.7,A -85,B 0,C 180,E1 -21254.828,E2 -21254.828} C_VEL
LIN {X 0,Y 232.357,Z 719.484,A -85,B 0,C 180,E1 -21257.606,E2 -21257.606} C_VEL
LIN {X 0,Y 237.779,Z 710.743,A -85,B 0,C 180,E1 -21259.872,E2 -21259.872} C_VEL
LIN {X 0,Y 242.341,Z 702.427,A -85,B 0,C 180,E1 -21261.613,E2 -21261.613} C_VEL
LIN {X 0,Y 243.441,Z 698.129,A -85,B 0,C 180,E1 -21262.938,E2 -21262.938} C_VEL
LIN {X 0,Y 244.584,Z 689.689,A -85,B 0,C 180,E1 -21265.892,E2 -21265.892} C_VEL
LIN {X 0,Y 245.205,Z 682.424,A -85,B 0,C 180,E1 -21268.737,E2 -21268.737} C_VEL
LIN {X 0,Y 245.276,Z 680.431,A -85,B 0,C 180,E1 -21269.672,E2 -21269.672} C_VEL
LIN {X 0,Y 244.989,Z 677.076,A -85,B 0,C 180,E1 -21271.924,E2 -21271.924} C_VEL
LIN {X 0,Y 244.868,Z 675.706,A -85,B 0,C 180,E1 -21273.047,E2 -21273.047} C_VEL
LIN {X 0,Y 244.767,Z 673.25,A -85,B 0,C 180,E1 -21277.084,E2 -21277.084} C_VEL
LIN {X 0,Y 245.056,Z 673.146,A -85,B 0,C 180,E1 -21279.258,E2 -21279.258} C_VEL
LIN {X 0,Y 245.376,Z 674.207,A -85,B 0,C 180,E1 -21281.206,E2 -21281.206} C_VEL
LIN {X 0,Y 245.965,Z 678.433,A -85,B 0,C 180,E1 -21284.415,E2 -21284.415} C_VEL
LIN {X 0,Y 245.962,Z 679.797,A -85,B 0,C 180,E1 -21285.034,E2 -21285.034} C_VEL
LIN {X 0,Y 244.898,Z 688.663,A -85,B 0,C 180,E1 -21287.75,E2 -21287.75} C_VEL
LIN {X 0,Y 243.404,Z 697.651,A -85,B 0,C 180,E1 -21290.095,E2 -21290.095} C_VEL
LIN {X 0,Y 241.224,Z 706.76,A -85,B 0,C 180,E1 -21292.28,E2 -21292.28} C_VEL
LIN {X 0,Y 238.607,Z 714.2,A -85,B 0,C 180,E1 -21293.91,E2 -21293.91} C_VEL
LIN {X 0,Y 233.43,Z 725.032,A -85,B 0,C 180,E1 -21296.231,E2 -21296.231} C_VEL
LIN {X 0,Y 230.833,Z 729.13,A -85,B 0,C 180,E1 -21297.093,E2 -21297.093} C_VEL
LIN {X 0,Y 225.038,Z 735.666,A -85,B 0,C 180,E1 -21298.294,E2 -21298.294} C_VEL
LIN {X 0,Y 219.053,Z 741.642,A -85,B 0,C 180,E1 -21299.625,E2 -21299.625} C_VEL
LIN {X 0,Y 216.211,Z 744.853,A -85,B 0,C 180,E1 -21300.685,E2 -21300.685} C_VEL
LIN {X 0,Y 211.607,Z 750.959,A -85,B 0,C 180,E1 -21303.363,E2 -21303.363} C_VEL
LIN {X 0,Y 206.805,Z 756.898,A -85,B 0,C 180,E1 -21306.773,E2 -21306.773} C_VEL
LIN {X 0,Y 203.685,Z 760.778,A -85,B 0,C 180,E1 -21309.818,E2 -21309.818} C_VEL
LIN {X 0,Y 200.543,Z 764.244,A -85,B 0,C 180,E1 -21313.72,E2 -21313.72} C_VEL
LIN {X 0,Y 198.59,Z 766.291,A -85,B 0,C 180,E1 -21317.743,E2 -21317.743} C_VEL
LIN {X 0,Y 197.713,Z 766.922,A -85,B 0,C 180,E1 -21321.828,E2 -21321.828} C_VEL
LIN {X 0,Y 197.733,Z 766.035,A -85,B 0,C 180,E1 -21325.926,E2 -21325.926} C_VEL
LIN {X 0,Y 198.244,Z 763.609,A -85,B 0,C 180,E1 -21330.002,E2 -21330.002} C_VEL
LIN {X 0,Y 198.04,Z 760.509,A -85,B 0,C 180,E1 -21333.053,E2 -21333.053} C_VEL
LIN {X 0,Y 198.097,Z 756.312,A -85,B 0,C 180,E1 -21336.112,E2 -21336.112} C_VEL
LIN {X 0,Y 198.339,Z 749.726,A -85,B 0,C 180,E1 -21339.692,E2 -21339.692} C_VEL
LIN {X 0,Y 198.963,Z 742.537,A -85,B 0,C 180,E1 -21342.756,E2 -21342.756} C_VEL
LIN {X 0,Y 199.869,Z 735.233,A -85,B 0,C 180,E1 -21345.293,E2 -21345.293} C_VEL
LIN {X 0,Y 201.233,Z 725.45,A -85,B 0,C 180,E1 -21348.058,E2 -21348.058} C_VEL
LIN {X 0,Y 202.698,Z 715.727,A -85,B 0,C 180,E1 -21350.289,E2 -21350.289} C_VEL
LIN {X 0,Y 203.534,Z 709.112,A -85,B 0,C 180,E1 -21351.58,E2 -21351.58} C_VEL
LIN {X 0,Y 203.634,Z 695.248,A -85,B 0,C 180,E1 -21353.926,E2 -21353.926} C_VEL
LIN {X 0,Y 203.925,Z 684.613,A -85,B 0,C 180,E1 -21356.061,E2 -21356.061} C_VEL
LIN {X 0,Y 203.989,Z 672.779,A -85,B 0,C 180,E1 -21357.998,E2 -21357.998} C_VEL
LIN {X 0,Y 203.594,Z 660.701,A -85,B 0,C 180,E1 -21359.604,E2 -21359.604} C_VEL
LIN {X 0,Y 202.624,Z 647.447,A -85,B 0,C 180,E1 -21360.992,E2 -21360.992} C_VEL
LIN {X 0,Y 201.153,Z 635.493,A -85,B 0,C 180,E1 -21361.968,E2 -21361.968} C_VEL
LIN {X 0,Y 201.222,Z 631.683,A -85,B 0,C 180,E1 -21362.895,E2 -21362.895} C_VEL
LIN {X 0,Y 203.413,Z 622.59,A -85,B 0,C 180,E1 -21368.457,E2 -21368.457} C_VEL
LIN {X 0,Y 203.7,Z 620.988,A -85,B 0,C 180,E1 -21369.445,E2 -21369.445} C_VEL
LIN {X 0,Y 203.092,Z 616.904,A -85,B 0,C 180,E1 -21372.17,E2 -21372.17} C_VEL
LIN {X 0,Y 201.658,Z 609.964,A -85,B 0,C 180,E1 -21377.046,E2 -21377.046} C_VEL
LIN {X 0,Y 200.433,Z 603.218,A -85,B 0,C 180,E1 -21382.147,E2 -21382.147} C_VEL
LIN {X 0,Y 199.726,Z 599.616,A -85,B 0,C 180,E1 -21385.045,E2 -21385.045} C_VEL
LIN {X 0,Y 199.711,Z 599.614,A -85,B 0,C 180,E1 -21388.138,E2 -21388.138} C_VEL
LIN {X 0,Y 199.693,Z 599.61,A -85,B 0,C 180,E1 -21392.772,E2 -21392.772} C_VEL
LIN {X 0,Y 199.745,Z 599.603,A -85,B 0,C 180,E1 -21397.229,E2 -21397.229} C_VEL
LIN {X 0,Y 199.803,Z 599.599,A -85,B 0,C 180,E1 -21401.757,E2 -21401.757} C_VEL
LIN {X 0,Y 199.854,Z 599.593,A -85,B 0,C 180,E1 -21405.749,E2 -21405.749} C_VEL
LIN {X 0,Y 200.082,Z 599.564,A -85,B 0,C 180,E1 -21409.884,E2 -21409.884} C_VEL
LIN {X 0,Y 200.138,Z 599.554,A -85,B 0,C 180,E1 -21411.925,E2 -21411.925} C_VEL
LIN {X 0,Y 200.327,Z 599.53,A -85,B 0,C 180,E1 -21417.989,E2 -21417.989} C_VEL
LIN {X 0,Y 200.485,Z 599.512,A -85,B 0,C 180,E1 -21419.999,E2 -21419.999} C_VEL
LIN {X 0,Y 200.034,Z 599.551,A -85,B 0,C 180,E1 -21424.029,E2 -21424.029} C_VEL
LIN {X 0,Y 200.117,Z 599.552,A -85,B 0,C 180,E1 -21428.075,E2 -21428.075} C_VEL
LIN {X 0,Y 199.918,Z 599.581,A -85,B 0,C 180,E1 -21432.176,E2 -21432.176} C_VEL
LIN {X 0,Y 199.808,Z 599.578,A -85,B 0,C 180,E1 -21436.342,E2 -21436.342} C_VEL
LIN {X 0,Y 199.705,Z 599.61,A -85,B 0,C 180,E1 -21440.604,E2 -21440.604} C_VEL
LIN {X 0,Y 199.677,Z 599.602,A -85,B 0,C 180,E1 -21444.983,E2 -21444.983} C_VEL
LIN {X 0,Y 199.679,Z 599.607,A -85,B 0,C 180,E1 -21449.521,E2 -21449.521} C_VEL
LIN {X 0,Y 199.681,Z 599.613,A -85,B 0,C 180,E1 -21452.357,E2 -21452.357} C_VEL
LIN {X 0,Y 199.626,Z 599.618,A -85,B 0,C 180,E1 -21456.761,E2 -21456.761} C_VEL
LIN {X 0,Y 199.611,Z 599.617,A -85,B 0,C 180,E1 -21459.326,E2 -21459.326} C_VEL
LIN {X 0,Y 199.578,Z 599.622,A -85,B 0,C 180,E1 -21462.309,E2 -21462.309} C_VEL
LIN {X 0,Y 199.614,Z 599.607,A -85,B 0,C 180,E1 -21465.236,E2 -21465.236} C_VEL
LIN {X 0,Y 199.624,Z 599.616,A -85,B 0,C 180,E1 -21468.014,E2 -21468.014} C_VEL
LIN {X 0,Y 199.644,Z 599.609,A -85,B 0,C 180,E1 -21470.754,E2 -21470.754} C_VEL
LIN {X 0,Y 199.635,Z 599.616,A -85,B 0,C 180,E1 -21475.716,E2 -21475.716} C_VEL
LIN {X 0,Y 199.698,Z 599.603,A -85,B 0,C 180,E1 -21478.135,E2 -21478.135} C_VEL
LIN {X 0,Y 199.686,Z 599.606,A -85,B 0,C 180,E1 -21482.77,E2 -21482.77} C_VEL
LIN {X 0,Y 199.739,Z 599.601,A -85,B 0,C 180,E1 -21487.227,E2 -21487.227} C_VEL
LIN {X 0,Y 199.813,Z 599.594,A -85,B 0,C 180,E1 -21492.709,E2 -21492.709} C_VEL
LIN {X 0,Y 199.826,Z 599.733,A -85,B 0,C 180,E1 -21493.42,E2 -21493.42} C_VEL
LIN {X 0,Y 201.719,Z 604.613,A -85,B 0,C 180,E1 -21494.205,E2 -21494.205} C_VEL
LIN {X 0,Y 205.902,Z 615.529,A -85,B 0,C 180,E1 -21496.175,E2 -21496.175} C_VEL
LIN {X 0,Y 208.807,Z 624.97,A -85,B 0,C 180,E1 -21498.063,E2 -21498.063} C_VEL
LIN {X 0,Y 210.456,Z 632.692,A -85,B 0,C 180,E1 -21499.743,E2 -21499.743} C_VEL
LIN {X 0,Y 208.588,Z 643.598,A -85,B 0,C 180,E1 -21502.009,E2 -21502.009} C_VEL
LIN {X 0,Y 206.565,Z 653.522,A -85,B 0,C 180,E1 -21504.63,E2 -21504.63} C_VEL
LIN {X 0,Y 204.74,Z 662.266,A -85,B 0,C 180,E1 -21507.539,E2 -21507.539} C_VEL
LIN {X 0,Y 203.229,Z 669.283,A -85,B 0,C 180,E1 -21510.494,E2 -21510.494} C_VEL
LIN {X 0,Y 201.761,Z 675.756,A -85,B 0,C 180,E1 -21513.993,E2 -21513.993} C_VEL
LIN {X 0,Y 200.921,Z 680.039,A -85,B 0,C 180,E1 -21517.03,E2 -21517.03} C_VEL
LIN {X 0,Y 200.471,Z 683.26,A -85,B 0,C 180,E1 -21520.093,E2 -21520.093} C_VEL
LIN {X 0,Y 200.37,Z 684.885,A -85,B 0,C 180,E1 -21522.147,E2 -21522.147} C_VEL
LIN {X 0,Y 200.442,Z 686.054,A -85,B 0,C 180,E1 -21524.206,E2 -21524.206} C_VEL
LIN {X 0,Y 201.139,Z 687.191,A -85,B 0,C 180,E1 -21528.327,E2 -21528.327} C_VEL
LIN {X 0,Y 201.736,Z 687.165,A -85,B 0,C 180,E1 -21530.386,E2 -21530.386} C_VEL
LIN {X 0,Y 202.493,Z 686.695,A -85,B 0,C 180,E1 -21532.442,E2 -21532.442} C_VEL
LIN {X 0,Y 203.514,Z 685.816,A -85,B 0,C 180,E1 -21534.479,E2 -21534.479} C_VEL
LIN {X 0,Y 204.929,Z 684.208,A -85,B 0,C 180,E1 -21536.919,E2 -21536.919} C_VEL
LIN {X 0,Y 207.561,Z 680.544,A -85,B 0,C 180,E1 -21540.522,E2 -21540.522} C_VEL
LIN {X 0,Y 210.31,Z 676.1,A -85,B 0,C 180,E1 -21543.569,E2 -21543.569} C_VEL
LIN {X 0,Y 213.285,Z 670.681,A -85,B 0,C 180,E1 -21546.376,E2 -21546.376} C_VEL
LIN {X 0,Y 216.721,Z 663.665,A -85,B 0,C 180,E1 -21549.169,E2 -21549.169} C_VEL
LIN {X 0,Y 219.296,Z 657.925,A -85,B 0,C 180,E1 -21551.012,E2 -21551.012} C_VEL
LIN {X 0,Y 219.335,Z 656.604,A -85,B 0,C 180,E1 -21551.507,E2 -21551.507} C_VEL
LIN {X 0,Y 213.356,Z 651.321,A -85,B 0,C 180,E1 -21554.911,E2 -21554.911} C_VEL
LIN {X 0,Y 207.072,Z 646.346,A -85,B 0,C 180,E1 -21558.3,E2 -21558.3} C_VEL
LIN {X 0,Y 204.469,Z 645.902,A -85,B 0,C 180,E1 -21559.228,E2 -21559.228} C_VEL
LIN {X 0,Y 202.544,Z 644.928,A -85,B 0,C 180,E1 -21560.138,E2 -21560.138} C_VEL
LIN {X 0,Y 204.836,Z 660.756,A -85,B 0,C 180,E1 -21561.861,E2 -21561.861} C_VEL
LIN {X 0,Y 206.294,Z 671.973,A -85,B 0,C 180,E1 -21563.404,E2 -21563.404} C_VEL
LIN {X 0,Y 204.715,Z 683.536,A -85,B 0,C 180,E1 -21565.199,E2 -21565.199} C_VEL
LIN {X 0,Y 202.922,Z 695.536,A -85,B 0,C 180,E1 -21567.533,E2 -21567.533} C_VEL
LIN {X 0,Y 201.307,Z 706.34,A -85,B 0,C 180,E1 -21570.167,E2 -21570.167} C_VEL
LIN {X 0,Y 199.93,Z 715.197,A -85,B 0,C 180,E1 -21572.808,E2 -21572.808} C_VEL
LIN {X 0,Y 198.808,Z 723.831,A -85,B 0,C 180,E1 -21576.015,E2 -21576.015} C_VEL
LIN {X 0,Y 198.042,Z 730.759,A -85,B 0,C 180,E1 -21579.215,E2 -21579.215} C_VEL
LIN {X 0,Y 197.546,Z 736.236,A -85,B 0,C 180,E1 -21582.399,E2 -21582.399} C_VEL
LIN {X 0,Y 197.314,Z 740.481,A -85,B 0,C 180,E1 -21585.563,E2 -21585.563} C_VEL
LIN {X 0,Y 197.317,Z 742.694,A -85,B 0,C 180,E1 -21587.661,E2 -21587.661} C_VEL
LIN {X 0,Y 197.564,Z 744.482,A -85,B 0,C 180,E1 -21589.755,E2 -21589.755} C_VEL
LIN {X 0,Y 198.289,Z 746.381,A -85,B 0,C 180,E1 -21592.917,E2 -21592.917} C_VEL
LIN {X 0,Y 199.276,Z 747.352,A -85,B 0,C 180,E1 -21595.956,E2 -21595.956} C_VEL
LIN {X 0,Y 201.388,Z 747.357,A -85,B 0,C 180,E1 -21600.001,E2 -21600.001} C_VEL
LIN {X 0,Y 204.416,Z 745.812,A -85,B 0,C 180,E1 -21603.944,E2 -21603.944} C_VEL
LIN {X 0,Y 208.364,Z 742.787,A -85,B 0,C 180,E1 -21607.755,E2 -21607.755} C_VEL
LIN {X 0,Y 211.986,Z 739.456,A -85,B 0,C 180,E1 -21610.507,E2 -21610.507} C_VEL
LIN {X 0,Y 217.014,Z 734.064,A -85,B 0,C 180,E1 -21613.709,E2 -21613.709} C_VEL
LIN {X 0,Y 222.354,Z 727.709,A -85,B 0,C 180,E1 -21616.528,E2 -21616.528} C_VEL
LIN {X 0,Y 227.633,Z 720.688,A -85,B 0,C 180,E1 -21618.917,E2 -21618.917} C_VEL
LIN {X 0,Y 233.351,Z 712.168,A -85,B 0,C 180,E1 -21621.188,E2 -21621.188} C_VEL
LIN {X 0,Y 237.369,Z 705.543,A -85,B 0,C 180,E1 -21622.638,E2 -21622.638} C_VEL
LIN {X 0,Y 238.338,Z 702.797,A -85,B 0,C 180,E1 -21623.46,E2 -21623.46} C_VEL
LIN {X 0,Y 239.901,Z 695.715,A -85,B 0,C 180,E1 -21626.068,E2 -21626.068} C_VEL
LIN {X 0,Y 241.174,Z 688.372,A -85,B 0,C 180,E1 -21629.051,E2 -21629.051} C_VEL
LIN {X 0,Y 241.494,Z 685.185,A -85,B 0,C 180,E1 -21630.718,E2 -21630.718} C_VEL
LIN {X 0,Y 241.475,Z 682.867,A -85,B 0,C 180,E1 -21632.436,E2 -21632.436} C_VEL
LIN {X 0,Y 241.509,Z 681.716,A -85,B 0,C 180,E1 -21633.567,E2 -21633.567} C_VEL
LIN {X 0,Y 241.416,Z 680.42,A -85,B 0,C 180,E1 -21635.608,E2 -21635.608} C_VEL
LIN {X 0,Y 241.794,Z 679.555,A -85,B 0,C 180,E1 -21638.302,E2 -21638.302} C_VEL
LIN {X 0,Y 242.044,Z 679.809,A -85,B 0,C 180,E1 -21639.703,E2 -21639.703} C_VEL
LIN {X 0,Y 242.226,Z 680.594,A -85,B 0,C 180,E1 -21641.033,E2 -21641.033} C_VEL
LIN {X 0,Y 242.419,Z 683.726,A -85,B 0,C 180,E1 -21643.552,E2 -21643.552} C_VEL
LIN {X 0,Y 242.456,Z 684.651,A -85,B 0,C 180,E1 -21644.082,E2 -21644.082} C_VEL
LIN {X 0,Y 241.705,Z 688.71,A -85,B 0,C 180,E1 -21645.498,E2 -21645.498} C_VEL
LIN {X 0,Y 240.209,Z 696.123,A -85,B 0,C 180,E1 -21647.709,E2 -21647.709} C_VEL
LIN {X 0,Y 237.738,Z 705.612,A -85,B 0,C 180,E1 -21650.23,E2 -21650.23} C_VEL
LIN {X 0,Y 235.122,Z 713.058,A -85,B 0,C 180,E1 -21652.043,E2 -21652.043} C_VEL
LIN {X 0,Y 231.511,Z 720.677,A -85,B 0,C 180,E1 -21653.706,E2 -21653.706} C_VEL
LIN {X 0,Y 225.364,Z 731.488,A -85,B 0,C 180,E1 -21656.392,E2 -21656.392} C_VEL
LIN {X 0,Y 220.214,Z 739.443,A -85,B 0,C 180,E1 -21658.763,E2 -21658.763} C_VEL
LIN {X 0,Y 216.211,Z 744.853,A -85,B 0,C 180,E1 -21660.685,E2 -21660.685} C_VEL
LIN {X 0,Y 213.385,Z 747.94,A -85,B 0,C 180,E1 -21661.819,E2 -21661.819} C_VEL
LIN {X 0,Y 207.381,Z 752.632,A -85,B 0,C 180,E1 -21663.568,E2 -21663.568} C_VEL
LIN {X 0,Y 201.622,Z 756.621,A -85,B 0,C 180,E1 -21665.51,E2 -21665.51} C_VEL
LIN {X 0,Y 199.232,Z 758.607,A -85,B 0,C 180,E1 -21666.922,E2 -21666.922} C_VEL
LIN {X 0,Y 195.272,Z 762.767,A -85,B 0,C 180,E1 -21671.102,E2 -21671.102} C_VEL
LIN {X 0,Y 192.466,Z 765.272,A -85,B 0,C 180,E1 -21675.192,E2 -21675.192} C_VEL
LIN {X 0,Y 191.029,Z 766.329,A -85,B 0,C 180,E1 -21679.402,E2 -21679.402} C_VEL
LIN {X 0,Y 190.575,Z 765.963,A -85,B 0,C 180,E1 -21683.65,E2 -21683.65} C_VEL
LIN {X 0,Y 190.672,Z 765.247,A -85,B 0,C 180,E1 -21685.774,E2 -21685.774} C_VEL
LIN {X 0,Y 190.802,Z 764.131,A -85,B 0,C 180,E1 -21687.891,E2 -21687.891} C_VEL
LIN {X 0,Y 191.208,Z 762.576,A -85,B 0,C 180,E1 -21690.002,E2 -21690.002} C_VEL
LIN {X 0,Y 191.018,Z 759.28,A -85,B 0,C 180,E1 -21693.166,E2 -21693.166} C_VEL
LIN {X 0,Y 191.108,Z 754.079,A -85,B 0,C 180,E1 -21696.813,E2 -21696.813} C_VEL
LIN {X 0,Y 191.37,Z 748.059,A -85,B 0,C 180,E1 -21700.048,E2 -21700.048} C_VEL
LIN {X 0,Y 192.06,Z 740.617,A -85,B 0,C 180,E1 -21703.223,E2 -21703.223} C_VEL
LIN {X 0,Y 193.286,Z 731.338,A -85,B 0,C 180,E1 -21706.369,E2 -21706.369} C_VEL
LIN {X 0,Y 194.831,Z 720.757,A -85,B 0,C 180,E1 -21709.22,E2 -21709.22} C_VEL
LIN {X 0,Y 196.457,Z 709.981,A -85,B 0,C 180,E1 -21711.545,E2 -21711.545} C_VEL
LIN {X 0,Y 196.563,Z 697.914,A -85,B 0,C 180,E1 -21713.72,E2 -21713.72} C_VEL
LIN {X 0,Y 197.006,Z 686.717,A -85,B 0,C 180,E1 -21716.196,E2 -21716.196} C_VEL
LIN {X 0,Y 197.201,Z 675.787,A -85,B 0,C 180,E1 -21718.18,E2 -21718.18} C_VEL
LIN {X 0,Y 197.017,Z 663.755,A -85,B 0,C 180,E1 -21719.963,E2 -21719.963} C_VEL
LIN {X 0,Y 196.192,Z 649.963,A -85,B 0,C 180,E1 -21721.57,E2 -21721.57} C_VEL
LIN {X 0,Y 194.746,Z 636.882,A -85,B 0,C 180,E1 -21722.755,E2 -21722.755} C_VEL
LIN {X 0,Y 194.299,Z 633.772,A -85,B 0,C 180,E1 -21723.03,E2 -21723.03} C_VEL
LIN {X 0,Y 194.412,Z 630.951,A -85,B 0,C 180,E1 -21723.75,E2 -21723.75} C_VEL
LIN {X 0,Y 196.434,Z 622.882,A -85,B 0,C 180,E1 -21728.873,E2 -21728.873} C_VEL
LIN {X 0,Y 196.58,Z 621.07,A -85,B 0,C 180,E1 -21730.057,E2 -21730.057} C_VEL
LIN {X 0,Y 195.546,Z 615.378,A -85,B 0,C 180,E1 -21734.043,E2 -21734.043} C_VEL
LIN {X 0,Y 194.115,Z 608.134,A -85,B 0,C 180,E1 -21739.494,E2 -21739.494} C_VEL
LIN {X 0,Y 192.979,Z 602.102,A -85,B 0,C 180,E1 -21744.359,E2 -21744.359} C_VEL
LIN {X 0,Y 192.625,Z 600.5,A -85,B 0,C 180,E1 -21745.877,E2 -21745.877} C_VEL
LIN {X 0,Y 192.657,Z 600.487,A -85,B 0,C 180,E1 -21751.108,E2 -21751.108} C_VEL
LIN {X 0,Y 192.713,Z 600.482,A -85,B 0,C 180,E1 -21756.349,E2 -21756.349} C_VEL
LIN {X 0,Y 192.739,Z 600.478,A -85,B 0,C 180,E1 -21761.457,E2 -21761.457} C_VEL
LIN {X 0,Y 192.778,Z 600.474,A -85,B 0,C 180,E1 -21765.214,E2 -21765.214} C_VEL
LIN {X 0,Y 193.027,Z 600.442,A -85,B 0,C 180,E1 -21769.51,E2 -21769.51} C_VEL
LIN {X 0,Y 193.01,Z 600.442,A -85,B 0,C 180,E1 -21773.728,E2 -21773.728} C_VEL
LIN {X 0,Y 193.269,Z 600.409,A -85,B 0,C 180,E1 -21777.915,E2 -21777.915} C_VEL
LIN {X 0,Y 193.449,Z 600.388,A -85,B 0,C 180,E1 -21779.999,E2 -21779.999} C_VEL
LIN {X 0,Y 192.98,Z 600.427,A -85,B 0,C 180,E1 -21784.176,E2 -21784.176} C_VEL
LIN {X 0,Y 193.068,Z 600.432,A -85,B 0,C 180,E1 -21788.372,E2 -21788.372} C_VEL
LIN {X 0,Y 192.857,Z 600.457,A -85,B 0,C 180,E1 -21792.629,E2 -21792.629} C_VEL
LIN {X 0,Y 192.762,Z 600.458,A -85,B 0,C 180,E1 -21796.957,E2 -21796.957} C_VEL
LIN {X 0,Y 192.641,Z 600.487,A -85,B 0,C 180,E1 -21801.396,E2 -21801.396} C_VEL
LIN {X 0,Y 192.669,Z 600.479,A -85,B 0,C 180,E1 -21804.223,E2 -21804.223} C_VEL
LIN {X 0,Y 192.654,Z 600.481,A -85,B 0,C 180,E1 -21808.891,E2 -21808.891} C_VEL
LIN {X 0,Y 192.602,Z 600.49,A -85,B 0,C 180,E1 -21813.184,E2 -21813.184} C_VEL
LIN {X 0,Y 192.554,Z 600.497,A -85,B 0,C 180,E1 -21818.35,E2 -21818.35} C_VEL
LIN {X 0,Y 192.519,Z 600.497,A -85,B 0,C 180,E1 -21823.102,E2 -21823.102} C_VEL
LIN {X 0,Y 192.549,Z 600.495,A -85,B 0,C 180,E1 -21826.885,E2 -21826.885} C_VEL
LIN {X 0,Y 192.577,Z 600.487,A -85,B 0,C 180,E1 -21831.652,E2 -21831.652} C_VEL
LIN {X 0,Y 192.6,Z 600.491,A -85,B 0,C 180,E1 -21834.277,E2 -21834.277} C_VEL
LIN {X 0,Y 192.601,Z 600.49,A -85,B 0,C 180,E1 -21839.277,E2 -21839.277} C_VEL
LIN {X 0,Y 192.662,Z 600.486,A -85,B 0,C 180,E1 -21841.689,E2 -21841.689} C_VEL
LIN {X 0,Y 192.707,Z 600.479,A -85,B 0,C 180,E1 -21846.347,E2 -21846.347} C_VEL
LIN {X 0,Y 192.79,Z 600.608,A -85,B 0,C 180,E1 -21852.406,E2 -21852.406} C_VEL
LIN {X 0,Y 195.065,Z 606.32,A -85,B 0,C 180,E1 -21853.384,E2 -21853.384} C_VEL
LIN {X 0,Y 199.097,Z 616.909,A -85,B 0,C 180,E1 -21855.406,E2 -21855.406} C_VEL
LIN {X 0,Y 202.131,Z 626.683,A -85,B 0,C 180,E1 -21857.471,E2 -21857.471} C_VEL
LIN {X 0,Y 203.587,Z 632.873,A -85,B 0,C 180,E1 -21858.894,E2 -21858.894} C_VEL
LIN {X 0,Y 203.687,Z 634.68,A -85,B 0,C 180,E1 -21859.288,E2 -21859.288} C_VEL
LIN {X 0,Y 201.822,Z 644.821,A -85,B 0,C 180,E1 -21861.487,E2 -21861.487} C_VEL
LIN {X 0,Y 199.882,Z 653.902,A -85,B 0,C 180,E1 -21863.943,E2 -21863.943} C_VEL
LIN {X 0,Y 197.962,Z 662.749,A -85,B 0,C 180,E1 -21866.946,E2 -21866.946} C_VEL
LIN {X 0,Y 196.376,Z 669.892,A -85,B 0,C 180,E1 -21869.998,E2 -21869.998} C_VEL
LIN {X 0,Y 195.013,Z 675.629,A -85,B 0,C 180,E1 -21873.097,E2 -21873.097} C_VEL
LIN {X 0,Y 194.044,Z 680.168,A -85,B 0,C 180,E1 -21876.236,E2 -21876.236} C_VEL
LIN {X 0,Y 193.663,Z 682.572,A -85,B 0,C 180,E1 -21878.344,E2 -21878.344} C_VEL
LIN {X 0,Y 193.368,Z 685.056,A -85,B 0,C 180,E1 -21881.097,E2 -21881.097} C_VEL
LIN {X 0,Y 193.474,Z 687.205,A -85,B 0,C 180,E1 -21884.729,E2 -21884.729} C_VEL
LIN {X 0,Y 194.265,Z 688.25,A -85,B 0,C 180,E1 -21889,E2 -21889} C_VEL
LIN {X 0,Y 194.947,Z 688.129,A -85,B 0,C 180,E1 -21891.129,E2 -21891.129} C_VEL
LIN {X 0,Y 195.809,Z 687.607,A -85,B 0,C 180,E1 -21893.252,E2 -21893.252} C_VEL
LIN {X 0,Y 196.902,Z 686.684,A -85,B 0,C 180,E1 -21895.358,E2 -21895.358} C_VEL
LIN {X 0,Y 198.267,Z 685.193,A -85,B 0,C 180,E1 -21897.605,E2 -21897.605} C_VEL
LIN {X 0,Y 200.444,Z 682.413,A -85,B 0,C 180,E1 -21900.555,E2 -21900.555} C_VEL
LIN {X 0,Y 203.619,Z 677.649,A -85,B 0,C 180,E1 -21904.07,E2 -21904.07} C_VEL
LIN {X 0,Y 206.846,Z 672.103,A -85,B 0,C 180,E1 -21907.089,E2 -21907.089} C_VEL
LIN {X 0,Y 210.432,Z 665.245,A -85,B 0,C 180,E1 -21909.944,E2 -21909.944} C_VEL
LIN {X 0,Y 212.491,Z 660.907,A -85,B 0,C 180,E1 -21911.411,E2 -21911.411} C_VEL
LIN {X 0,Y 211.895,Z 659.266,A -85,B 0,C 180,E1 -21912.263,E2 -21912.263} C_VEL
LIN {X 0,Y 207.827,Z 655.745,A -85,B 0,C 180,E1 -21914.754,E2 -21914.754} C_VEL
LIN {X 0,Y 204.557,Z 653.345,A -85,B 0,C 180,E1 -21916.597,E2 -21916.597} C_VEL
LIN {X 0,Y 201.023,Z 651.377,A -85,B 0,C 180,E1 -21918.375,E2 -21918.375} C_VEL
LIN {X 0,Y 196.614,Z 650.986,A -85,B 0,C 180,E1 -21919.954,E2 -21919.954} C_VEL
LIN {X 0,Y 196.252,Z 650.536,A -85,B 0,C 180,E1 -21920.242,E2 -21920.242} C_VEL
LIN {X 0,Y 198.236,Z 664.5,A -85,B 0,C 180,E1 -21921.948,E2 -21921.948} C_VEL
LIN {X 0,Y 199.227,Z 672.721,A -85,B 0,C 180,E1 -21923.153,E2 -21923.153} C_VEL
LIN {X 0,Y 197.385,Z 685.697,A -85,B 0,C 180,E1 -21925.272,E2 -21925.272} C_VEL
LIN {X 0,Y 195.643,Z 697.308,A -85,B 0,C 180,E1 -21927.701,E2 -21927.701} C_VEL
LIN {X 0,Y 194.032,Z 707.62,A -85,B 0,C 180,E1 -21930.373,E2 -21930.373} C_VEL
LIN {X 0,Y 192.556,Z 717.157,A -85,B 0,C 180,E1 -21933.443,E2 -21933.443} C_VEL
LIN {X 0,Y 191.558,Z 724.938,A -85,B 0,C 180,E1 -21936.516,E2 -21936.516} C_VEL
LIN {X 0,Y 190.879,Z 731.162,A -85,B 0,C 180,E1 -21939.527,E2 -21939.527} C_VEL
LIN {X 0,Y 190.411,Z 736.656,A -85,B 0,C 180,E1 -21942.827,E2 -21942.827} C_VEL
LIN {X 0,Y 190.219,Z 740.886,A -85,B 0,C 180,E1 -21946.105,E2 -21946.105} C_VEL
LIN {X 0,Y 190.392,Z 744.066,A -85,B 0,C 180,E1 -21949.365,E2 -21949.365} C_VEL
LIN {X 0,Y 191.374,Z 746.815,A -85,B 0,C 180,E1 -21953.676,E2 -21953.676} C_VEL
LIN {X 0,Y 192.987,Z 748.027,A -85,B 0,C 180,E1 -21957.914,E2 -21957.914} C_VEL
LIN {X 0,Y 195.626,Z 747.68,A -85,B 0,C 180,E1 -21962.06,E2 -21962.06} C_VEL
LIN {X 0,Y 199.182,Z 745.901,A -85,B 0,C 180,E1 -21966.077,E2 -21966.077} C_VEL
LIN {X 0,Y 203.737,Z 742.555,A -85,B 0,C 180,E1 -21969.933,E2 -21969.933} C_VEL
LIN {X 0,Y 209.302,Z 737.615,A -85,B 0,C 180,E1 -21973.595,E2 -21973.595} C_VEL
LIN {X 0,Y 214.016,Z 732.747,A -85,B 0,C 180,E1 -21976.209,E2 -21976.209} C_VEL
LIN {X 0,Y 220.253,Z 725.548,A -85,B 0,C 180,E1 -21979.091,E2 -21979.091} C_VEL
LIN {X 0,Y 226.001,Z 718.076,A -85,B 0,C 180,E1 -21981.432,E2 -21981.432} C_VEL
LIN {X 0,Y 232.22,Z 708.89,A -85,B 0,C 180,E1 -21983.642,E2 -21983.642} C_VEL
LIN {X 0,Y 233.149,Z 707.327,A -85,B 0,C 180,E1 -21984.015,E2 -21984.015} C_VEL
LIN {X 0,Y 235.194,Z 700.585,A -85,B 0,C 180,E1 -21986.631,E2 -21986.631} C_VEL
LIN {X 0,Y 236.998,Z 693.636,A -85,B 0,C 180,E1 -21989.623,E2 -21989.623} C_VEL
LIN {X 0,Y 237.509,Z 691.289,A -85,B 0,C 180,E1 -21990.897,E2 -21990.897} C_VEL
LIN {X 0,Y 237.724,Z 689.472,A -85,B 0,C 180,E1 -21992.151,E2 -21992.151} C_VEL
LIN {X 0,Y 237.928,Z 687.5,A -85,B 0,C 180,E1 -21994.204,E2 -21994.204} C_VEL
LIN {X 0,Y 238.22,Z 686.041,A -85,B 0,C 180,E1 -21997.201,E2 -21997.201} C_VEL
LIN {X 0,Y 238.437,Z 685.805,A -85,B 0,C 180,E1 -21998.243,E2 -21998.243} C_VEL
LIN {X 0,Y 238.712,Z 686.477,A -85,B 0,C 180,E1 -22000.37,E2 -22000.37} C_VEL
LIN {X 0,Y 238.754,Z 688.898,A -85,B 0,C 180,E1 -22002.619,E2 -22002.619} C_VEL
LIN {X 0,Y 238.75,Z 689.606,A -85,B 0,C 180,E1 -22003.156,E2 -22003.156} C_VEL
LIN {X 0,Y 238.198,Z 692.273,A -85,B 0,C 180,E1 -22004.233,E2 -22004.233} C_VEL
LIN {X 0,Y 235.968,Z 700.243,A -85,B 0,C 180,E1 -22006.765,E2 -22006.765} C_VEL
LIN {X 0,Y 233.006,Z 709.1,A -85,B 0,C 180,E1 -22009.255,E2 -22009.255} C_VEL
LIN {X 0,Y 229.85,Z 716.68,A -85,B 0,C 180,E1 -22011.187,E2 -22011.187} C_VEL
LIN {X 0,Y 223.323,Z 727.925,A -85,B 0,C 180,E1 -22013.841,E2 -22013.841} C_VEL
LIN {X 0,Y 217.059,Z 737.337,A -85,B 0,C 180,E1 -22016.606,E2 -22016.606} C_VEL
LIN {X 0,Y 210.318,Z 745.918,A -85,B 0,C 180,E1 -22019.663,E2 -22019.663} C_VEL
LIN {X 0,Y 205.35,Z 751.849,A -85,B 0,C 180,E1 -22022.484,E2 -22022.484} C_VEL
LIN {X 0,Y 200.179,Z 757.565,A -85,B 0,C 180,E1 -22026.101,E2 -22026.101} C_VEL
LIN {X 0,Y 199.232,Z 758.607,A -85,B 0,C 180,E1 -22026.922,E2 -22026.922} C_VEL
LIN {X 0,Y 196.937,Z 760.426,A -85,B 0,C 180,E1 -22028.411,E2 -22028.411} C_VEL
LIN {X 0,Y 191.729,Z 762.859,A -85,B 0,C 180,E1 -22030.802,E2 -22030.802} C_VEL
LIN {X 0,Y 186.943,Z 764.523,A -85,B 0,C 180,E1 -22033.376,E2 -22033.376} C_VEL
LIN {X 0,Y 185.358,Z 765.141,A -85,B 0,C 180,E1 -22035.112,E2 -22035.112} C_VEL
LIN {X 0,Y 184.034,Z 765.827,A -85,B 0,C 180,E1 -22038.994,E2 -22038.994} C_VEL
LIN {X 0,Y 183.528,Z 765.245,A -85,B 0,C 180,E1 -22043.405,E2 -22043.405} C_VEL
LIN {X 0,Y 183.62,Z 764.376,A -85,B 0,C 180,E1 -22045.612,E2 -22045.612} C_VEL
LIN {X 0,Y 184.193,Z 761.489,A -85,B 0,C 180,E1 -22050.002,E2 -22050.002} C_VEL
LIN {X 0,Y 183.996,Z 758.013,A -85,B 0,C 180,E1 -22053.287,E2 -22053.287} C_VEL
LIN {X 0,Y 184.075,Z 753.36,A -85,B 0,C 180,E1 -22056.579,E2 -22056.579} C_VEL
LIN {X 0,Y 184.318,Z 747.391,A -85,B 0,C 180,E1 -22059.882,E2 -22059.882} C_VEL
LIN {X 0,Y 185.009,Z 739.89,A -85,B 0,C 180,E1 -22063.177,E2 -22063.177} C_VEL
LIN {X 0,Y 186.248,Z 730.63,A -85,B 0,C 180,E1 -22066.442,E2 -22066.442} C_VEL
LIN {X 0,Y 187.793,Z 720.059,A -85,B 0,C 180,E1 -22069.401,E2 -22069.401} C_VEL
LIN {X 0,Y 189.404,Z 709.473,A -85,B 0,C 180,E1 -22071.783,E2 -22071.783} C_VEL
LIN {X 0,Y 189.501,Z 700.303,A -85,B 0,C 180,E1 -22073.497,E2 -22073.497} C_VEL
LIN {X 0,Y 189.962,Z 689.924,A -85,B 0,C 180,E1 -22076.064,E2 -22076.064} C_VEL
LIN {X 0,Y 190.373,Z 677.812,A -85,B 0,C 180,E1 -22078.493,E2 -22078.493} C_VEL
LIN {X 0,Y 190.335,Z 665.257,A -85,B 0,C 180,E1 -22080.513,E2 -22080.513} C_VEL
LIN {X 0,Y 189.747,Z 652.462,A -85,B 0,C 180,E1 -22082.171,E2 -22082.171} C_VEL
LIN {X 0,Y 188.522,Z 639.328,A -85,B 0,C 180,E1 -22083.498,E2 -22083.498} C_VEL
LIN {X 0,Y 187.524,Z 632.071,A -85,B 0,C 180,E1 -22084.137,E2 -22084.137} C_VEL
LIN {X 0,Y 187.652,Z 630.101,A -85,B 0,C 180,E1 -22084.714,E2 -22084.714} C_VEL
LIN {X 0,Y 189.409,Z 623.463,A -85,B 0,C 180,E1 -22089.11,E2 -22089.11} C_VEL
LIN {X 0,Y 189.365,Z 620.451,A -85,B 0,C 180,E1 -22091.208,E2 -22091.208} C_VEL
LIN {X 0,Y 187.878,Z 613.415,A -85,B 0,C 180,E1 -22096.404,E2 -22096.404} C_VEL
LIN {X 0,Y 186.75,Z 607.21,A -85,B 0,C 180,E1 -22101.441,E2 -22101.441} C_VEL
LIN {X 0,Y 185.817,Z 602.584,A -85,B 0,C 180,E1 -22105.434,E2 -22105.434} C_VEL
LIN {X 0,Y 185.573,Z 601.378,A -85,B 0,C 180,E1 -22106.619,E2 -22106.619} C_VEL
LIN {X 0,Y 185.589,Z 601.368,A -85,B 0,C 180,E1 -22110.576,E2 -22110.576} C_VEL
LIN {X 0,Y 185.594,Z 601.367,A -85,B 0,C 180,E1 -22115.383,E2 -22115.383} C_VEL
LIN {X 0,Y 185.614,Z 601.367,A -85,B 0,C 180,E1 -22120.075,E2 -22120.075} C_VEL
LIN {X 0,Y 185.731,Z 601.353,A -85,B 0,C 180,E1 -22124.639,E2 -22124.639} C_VEL
LIN {X 0,Y 185.949,Z 601.323,A -85,B 0,C 180,E1 -22129.328,E2 -22129.328} C_VEL
LIN {X 0,Y 185.974,Z 601.319,A -85,B 0,C 180,E1 -22133.489,E2 -22133.489} C_VEL
LIN {X 0,Y 186.213,Z 601.287,A -85,B 0,C 180,E1 -22137.836,E2 -22137.836} C_VEL
LIN {X 0,Y 186.413,Z 601.265,A -85,B 0,C 180,E1 -22139.999,E2 -22139.999} C_VEL
LIN {X 0,Y 185.928,Z 601.304,A -85,B 0,C 180,E1 -22144.335,E2 -22144.335} C_VEL
LIN {X 0,Y 186.015,Z 601.312,A -85,B 0,C 180,E1 -22148.691,E2 -22148.691} C_VEL
LIN {X 0,Y 185.769,Z 601.337,A -85,B 0,C 180,E1 -22153.119,E2 -22153.119} C_VEL
LIN {X 0,Y 185.68,Z 601.35,A -85,B 0,C 180,E1 -22158.866,E2 -22158.866} C_VEL
LIN {X 0,Y 185.601,Z 601.367,A -85,B 0,C 180,E1 -22162.25,E2 -22162.25} C_VEL
LIN {X 0,Y 185.566,Z 601.353,A -85,B 0,C 180,E1 -22167.03,E2 -22167.03} C_VEL
LIN {X 0,Y 185.583,Z 601.363,A -85,B 0,C 180,E1 -22169.491,E2 -22169.491} C_VEL
LIN {X 0,Y 185.503,Z 601.376,A -85,B 0,C 180,E1 -22174.63,E2 -22174.63} C_VEL
LIN {X 0,Y 185.508,Z 601.375,A -85,B 0,C 180,E1 -22177.311,E2 -22177.311} C_VEL
LIN {X 0,Y 185.474,Z 601.381,A -85,B 0,C 180,E1 -22180.723,E2 -22180.723} C_VEL
LIN {X 0,Y 185.511,Z 601.365,A -85,B 0,C 180,E1 -22186.037,E2 -22186.037} C_VEL
LIN {X 0,Y 185.505,Z 601.375,A -85,B 0,C 180,E1 -22189.903,E2 -22189.903} C_VEL
LIN {X 0,Y 185.546,Z 601.362,A -85,B 0,C 180,E1 -22192.694,E2 -22192.694} C_VEL
LIN {X 0,Y 185.542,Z 601.365,A -85,B 0,C 180,E1 -22197.973,E2 -22197.973} C_VEL
LIN {X 0,Y 185.582,Z 601.369,A -85,B 0,C 180,E1 -22200.575,E2 -22200.575} C_VEL
LIN {X 0,Y 185.588,Z 601.367,A -85,B 0,C 180,E1 -22205.381,E2 -22205.381} C_VEL
LIN {X 0,Y 185.608,Z 601.363,A -85,B 0,C 180,E1 -22210.073,E2 -22210.073} C_VEL
LIN {X 0,Y 185.681,Z 601.356,A -85,B 0,C 180,E1 -22211.274,E2 -22211.274} C_VEL
LIN {X 0,Y 186.248,Z 603.321,A -85,B 0,C 180,E1 -22211.585,E2 -22211.585} C_VEL
LIN {X 0,Y 190.997,Z 614.575,A -85,B 0,C 180,E1 -22213.814,E2 -22213.814} C_VEL
LIN {X 0,Y 194.293,Z 624.311,A -85,B 0,C 180,E1 -22215.909,E2 -22215.909} C_VEL
LIN {X 0,Y 196.508,Z 632.649,A -85,B 0,C 180,E1 -22217.861,E2 -22217.861} C_VEL
LIN {X 0,Y 197.031,Z 635.589,A -85,B 0,C 180,E1 -22218.582,E2 -22218.582} C_VEL
LIN {X 0,Y 195.277,Z 645.026,A -85,B 0,C 180,E1 -22220.678,E2 -22220.678} C_VEL
LIN {X 0,Y 193.251,Z 654.268,A -85,B 0,C 180,E1 -22223.21,E2 -22223.21} C_VEL
LIN {X 0,Y 191.197,Z 663.227,A -85,B 0,C 180,E1 -22226.31,E2 -22226.31} C_VEL
LIN {X 0,Y 189.529,Z 670.462,A -85,B 0,C 180,E1 -22229.463,E2 -22229.463} C_VEL
LIN {X 0,Y 188.293,Z 675.407,A -85,B 0,C 180,E1 -22232.137,E2 -22232.137} C_VEL
LIN {X 0,Y 187.217,Z 680.219,A -85,B 0,C 180,E1 -22235.383,E2 -22235.383} C_VEL
LIN {X 0,Y 186.581,Z 683.921,A -85,B 0,C 180,E1 -22238.664,E2 -22238.664} C_VEL
LIN {X 0,Y 186.342,Z 686.153,A -85,B 0,C 180,E1 -22241.307,E2 -22241.307} C_VEL
LIN {X 0,Y 186.494,Z 688.361,A -85,B 0,C 180,E1 -22245.293,E2 -22245.293} C_VEL
LIN {X 0,Y 186.859,Z 689.032,A -85,B 0,C 180,E1 -22247.509,E2 -22247.509} C_VEL
LIN {X 0,Y 187.712,Z 689.244,A -85,B 0,C 180,E1 -22250.611,E2 -22250.611} C_VEL
LIN {X 0,Y 189.162,Z 688.522,A -85,B 0,C 180,E1 -22254.12,E2 -22254.12} C_VEL
LIN {X 0,Y 190.343,Z 687.54,A -85,B 0,C 180,E1 -22256.298,E2 -22256.298} C_VEL
LIN {X 0,Y 191.716,Z 686.085,A -85,B 0,C 180,E1 -22258.458,E2 -22258.458} C_VEL
LIN {X 0,Y 194.178,Z 683.072,A -85,B 0,C 180,E1 -22261.653,E2 -22261.653} C_VEL
LIN {X 0,Y 197.31,Z 678.609,A -85,B 0,C 180,E1 -22264.993,E2 -22264.993} C_VEL
LIN {X 0,Y 201.051,Z 672.516,A -85,B 0,C 180,E1 -22268.348,E2 -22268.348} C_VEL
LIN {X 0,Y 204.943,Z 665.327,A -85,B 0,C 180,E1 -22271.301,E2 -22271.301} C_VEL
LIN {X 0,Y 205.645,Z 663.975,A -85,B 0,C 180,E1 -22271.777,E2 -22271.777} C_VEL
LIN {X 0,Y 205.208,Z 662.492,A -85,B 0,C 180,E1 -22272.593,E2 -22272.593} C_VEL
LIN {X 0,Y 200.57,Z 658.881,A -85,B 0,C 180,E1 -22275.51,E2 -22275.51} C_VEL
LIN {X 0,Y 197.208,Z 656.892,A -85,B 0,C 180,E1 -22277.383,E2 -22277.383} C_VEL
LIN {X 0,Y 190.474,Z 656.248,A -85,B 0,C 180,E1 -22279.921,E2 -22279.921} C_VEL
LIN {X 0,Y 189.933,Z 655.669,A -85,B 0,C 180,E1 -22280.367,E2 -22280.367} C_VEL
LIN {X 0,Y 191.833,Z 669.902,A -85,B 0,C 180,E1 -22282.353,E2 -22282.353} C_VEL
LIN {X 0,Y 192.093,Z 674.022,A -85,B 0,C 180,E1 -22282.999,E2 -22282.999} C_VEL
LIN {X 0,Y 190.283,Z 686.116,A -85,B 0,C 180,E1 -22285.077,E2 -22285.077} C_VEL
LIN {X 0,Y 188.503,Z 697.665,A -85,B 0,C 180,E1 -22287.593,E2 -22287.593} C_VEL
LIN {X 0,Y 186.966,Z 707.38,A -85,B 0,C 180,E1 -22290.188,E2 -22290.188} C_VEL
LIN {X 0,Y 185.614,Z 715.996,A -85,B 0,C 180,E1 -22292.977,E2 -22292.977} C_VEL
LIN {X 0,Y 184.585,Z 723.729,A -85,B 0,C 180,E1 -22296.028,E2 -22296.028} C_VEL
LIN {X 0,Y 183.849,Z 730.467,A -85,B 0,C 180,E1 -22299.293,E2 -22299.293} C_VEL
LIN {X 0,Y 183.271,Z 737.235,A -85,B 0,C 180,E1 -22303.465,E2 -22303.465} C_VEL
LIN {X 0,Y 183.158,Z 742.413,A -85,B 0,C 180,E1 -22307.817,E2 -22307.817} C_VEL
LIN {X 0,Y 183.601,Z 745.303,A -85,B 0,C 180,E1 -22311.193,E2 -22311.193} C_VEL
LIN {X 0,Y 184.191,Z 746.719,A -85,B 0,C 180,E1 -22313.428,E2 -22313.428} C_VEL
LIN {X 0,Y 185.789,Z 748.34,A -85,B 0,C 180,E1 -22317.833,E2 -22317.833} C_VEL
LIN {X 0,Y 188.463,Z 748.484,A -85,B 0,C 180,E1 -22322.138,E2 -22322.138} C_VEL
LIN {X 0,Y 192.104,Z 747.153,A -85,B 0,C 180,E1 -22326.302,E2 -22326.302} C_VEL
LIN {X 0,Y 196.782,Z 744.323,A -85,B 0,C 180,E1 -22330.287,E2 -22330.287} C_VEL
LIN {X 0,Y 200.962,Z 741.193,A -85,B 0,C 180,E1 -22333.14,E2 -22333.14} C_VEL
LIN {X 0,Y 205.656,Z 737.097,A -85,B 0,C 180,E1 -22335.867,E2 -22335.867} C_VEL
LIN {X 0,Y 210.907,Z 732.009,A -85,B 0,C 180,E1 -22338.456,E2 -22338.456} C_VEL
LIN {X 0,Y 217.652,Z 724.589,A -85,B 0,C 180,E1 -22341.302,E2 -22341.302} C_VEL
LIN {X 0,Y 223.927,Z 716.759,A -85,B 0,C 180,E1 -22343.589,E2 -22343.589} C_VEL
LIN {X 0,Y 227.81,Z 711.395,A -85,B 0,C 180,E1 -22344.889,E2 -22344.889} C_VEL
LIN {X 0,Y 228.808,Z 709.541,A -85,B 0,C 180,E1 -22345.47,E2 -22345.47} C_VEL
LIN {X 0,Y 231.214,Z 703.213,A -85,B 0,C 180,E1 -22348.182,E2 -22348.182} C_VEL
LIN {X 0,Y 233.121,Z 697.628,A -85,B 0,C 180,E1 -22350.832,E2 -22350.832} C_VEL
LIN {X 0,Y 233.782,Z 694.917,A -85,B 0,C 180,E1 -22352.761,E2 -22352.761} C_VEL
LIN {X 0,Y 234.118,Z 693.221,A -85,B 0,C 180,E1 -22354.776,E2 -22354.776} C_VEL
LIN {X 0,Y 234.484,Z 692.289,A -85,B 0,C 180,E1 -22356.831,E2 -22356.831} C_VEL
LIN {X 0,Y 234.882,Z 692.105,A -85,B 0,C 180,E1 -22358.929,E2 -22358.929} C_VEL
LIN {X 0,Y 235.024,Z 693.376,A -85,B 0,C 180,E1 -22361.139,E2 -22361.139} C_VEL
LIN {X 0,Y 234.751,Z 695.621,A -85,B 0,C 180,E1 -22362.817,E2 -22362.817} C_VEL
LIN {X 0,Y 232.713,Z 701.543,A -85,B 0,C 180,E1 -22364.921,E2 -22364.921} C_VEL
LIN {X 0,Y 229.853,Z 708.975,A -85,B 0,C 180,E1 -22367.209,E2 -22367.209} C_VEL
LIN {X 0,Y 227.187,Z 715.026,A -85,B 0,C 180,E1 -22368.927,E2 -22368.927} C_VEL
LIN {X 0,Y 224.759,Z 719.675,A -85,B 0,C 180,E1 -22370.135,E2 -22370.135} C_VEL
LIN {X 0,Y 217.87,Z 730.19,A -85,B 0,C 180,E1 -22372.786,E2 -22372.786} C_VEL
LIN {X 0,Y 211.326,Z 739.115,A -85,B 0,C 180,E1 -22375.575,E2 -22375.575} C_VEL
LIN {X 0,Y 205.677,Z 745.634,A -85,B 0,C 180,E1 -22378.022,E2 -22378.022} C_VEL
LIN {X 0,Y 200.65,Z 751.12,A -85,B 0,C 180,E1 -22380.638,E2 -22380.638} C_VEL
LIN {X 0,Y 194.857,Z 756.915,A -85,B 0,C 180,E1 -22384.356,E2 -22384.356} C_VEL
LIN {X 0,Y 190.389,Z 761.235,A -85,B 0,C 180,E1 -22388.34,E2 -22388.34} C_VEL
LIN {X 0,Y 186.911,Z 764.097,A -85,B 0,C 180,E1 -22392.496,E2 -22392.496} C_VEL
LIN {X 0,Y 185.358,Z 765.141,A -85,B 0,C 180,E1 -22395.112,E2 -22395.112} C_VEL
LIN {X 0,Y 184.003,Z 765.597,A -85,B 0,C 180,E1 -22396.892,E2 -22396.892} C_VEL
LIN {X 0,Y 180.413,Z 765.516,A -85,B 0,C 180,E1 -22399.799,E2 -22399.799} C_VEL
LIN {X 0,Y 177.717,Z 764.88,A -85,B 0,C 180,E1 -22402.189,E2 -22402.189} C_VEL
LIN {X 0,Y 176.622,Z 764.119,A -85,B 0,C 180,E1 -22404.06,E2 -22404.06} C_VEL
LIN {X 0,Y 176.547,Z 763.817,A -85,B 0,C 180,E1 -22404.694,E2 -22404.694} C_VEL
LIN {X 0,Y 176.759,Z 762.107,A -85,B 0,C 180,E1 -22407.723,E2 -22407.723} C_VEL
LIN {X 0,Y 177.176,Z 760.331,A -85,B 0,C 180,E1 -22410.002,E2 -22410.002} C_VEL
LIN {X 0,Y 176.998,Z 756.642,A -85,B 0,C 180,E1 -22413.417,E2 -22413.417} C_VEL
LIN {X 0,Y 177.089,Z 751.223,A -85,B 0,C 180,E1 -22417.175,E2 -22417.175} C_VEL
LIN {X 0,Y 177.467,Z 744.378,A -85,B 0,C 180,E1 -22420.844,E2 -22420.844} C_VEL
LIN {X 0,Y 178.314,Z 736.284,A -85,B 0,C 180,E1 -22424.263,E2 -22424.263} C_VEL
LIN {X 0,Y 179.412,Z 728.041,A -85,B 0,C 180,E1 -22427.087,E2 -22427.087} C_VEL
LIN {X 0,Y 181.125,Z 717.044,A -85,B 0,C 180,E1 -22430.145,E2 -22430.145} C_VEL
LIN {X 0,Y 182.303,Z 708.416,A -85,B 0,C 180,E1 -22432.095,E2 -22432.095} C_VEL
LIN {X 0,Y 182.434,Z 701.99,A -85,B 0,C 180,E1 -22433.41,E2 -22433.41} C_VEL
LIN {X 0,Y 182.991,Z 691.621,A -85,B 0,C 180,E1 -22436.213,E2 -22436.213} C_VEL
LIN {X 0,Y 183.525,Z 679.627,A -85,B 0,C 180,E1 -22438.832,E2 -22438.832} C_VEL
LIN {X 0,Y 183.65,Z 667.357,A -85,B 0,C 180,E1 -22441.01,E2 -22441.01} C_VEL
LIN {X 0,Y 183.226,Z 653.918,A -85,B 0,C 180,E1 -22442.9,E2 -22442.9} C_VEL
LIN {X 0,Y 182.192,Z 641.061,A -85,B 0,C 180,E1 -22444.335,E2 -22444.335} C_VEL
LIN {X 0,Y 180.787,Z 630.138,A -85,B 0,C 180,E1 -22445.352,E2 -22445.352} C_VEL
LIN {X 0,Y 180.877,Z 629.39,A -85,B 0,C 180,E1 -22445.652,E2 -22445.652} C_VEL
LIN {X 0,Y 182.365,Z 623.722,A -85,B 0,C 180,E1 -22449.576,E2 -22449.576} C_VEL
LIN {X 0,Y 182.177,Z 620.605,A -85,B 0,C 180,E1 -22451.866,E2 -22451.866} C_VEL
LIN {X 0,Y 180.574,Z 613.157,A -85,B 0,C 180,E1 -22457.69,E2 -22457.69} C_VEL
LIN {X 0,Y 179.552,Z 607.287,A -85,B 0,C 180,E1 -22462.706,E2 -22462.706} C_VEL
LIN {X 0,Y 178.528,Z 602.254,A -85,B 0,C 180,E1 -22467.395,E2 -22467.395} C_VEL
LIN {X 0,Y 178.494,Z 602.253,A -85,B 0,C 180,E1 -22471.803,E2 -22471.803} C_VEL
LIN {X 0,Y 178.518,Z 602.249,A -85,B 0,C 180,E1 -22476.815,E2 -22476.815} C_VEL
LIN {X 0,Y 178.657,Z 602.233,A -85,B 0,C 180,E1 -22481.656,E2 -22481.656} C_VEL
LIN {X 0,Y 178.694,Z 602.23,A -85,B 0,C 180,E1 -22486.35,E2 -22486.35} C_VEL
LIN {X 0,Y 178.985,Z 602.19,A -85,B 0,C 180,E1 -22490.963,E2 -22490.963} C_VEL
LIN {X 0,Y 179.159,Z 602.166,A -85,B 0,C 180,E1 -22497.751,E2 -22497.751} C_VEL
LIN {X 0,Y 179.376,Z 602.141,A -85,B 0,C 180,E1 -22499.999,E2 -22499.999} C_VEL
LIN {X 0,Y 178.876,Z 602.181,A -85,B 0,C 180,E1 -22504.506,E2 -22504.506} C_VEL
LIN {X 0,Y 178.965,Z 602.191,A -85,B 0,C 180,E1 -22509.037,E2 -22509.037} C_VEL
LIN {X 0,Y 178.686,Z 602.218,A -85,B 0,C 180,E1 -22513.649,E2 -22513.649} C_VEL
LIN {X 0,Y 178.628,Z 602.23,A -85,B 0,C 180,E1 -22519.215,E2 -22519.215} C_VEL
LIN {X 0,Y 178.539,Z 602.233,A -85,B 0,C 180,E1 -22525.123,E2 -22525.123} C_VEL
LIN {X 0,Y 178.505,Z 602.25,A -85,B 0,C 180,E1 -22530.785,E2 -22530.785} C_VEL
LIN {X 0,Y 178.488,Z 602.248,A -85,B 0,C 180,E1 -22534.218,E2 -22534.218} C_VEL
LIN {X 0,Y 178.398,Z 602.26,A -85,B 0,C 180,E1 -22539.072,E2 -22539.072} C_VEL
LIN {X 0,Y 178.411,Z 602.26,A -85,B 0,C 180,E1 -22542.04,E2 -22542.04} C_VEL
LIN {X 0,Y 178.427,Z 602.244,A -85,B 0,C 180,E1 -22545.152,E2 -22545.152} C_VEL
LIN {X 0,Y 178.433,Z 602.257,A -85,B 0,C 180,E1 -22548.447,E2 -22548.447} C_VEL
LIN {X 0,Y 178.451,Z 602.251,A -85,B 0,C 180,E1 -22553.787,E2 -22553.787} C_VEL
LIN {X 0,Y 178.491,Z 602.248,A -85,B 0,C 180,E1 -22556.545,E2 -22556.545} C_VEL
LIN {X 0,Y 178.523,Z 602.246,A -85,B 0,C 180,E1 -22560.005,E2 -22560.005} C_VEL
LIN {X 0,Y 178.535,Z 602.246,A -85,B 0,C 180,E1 -22564.874,E2 -22564.874} C_VEL
LIN {X 0,Y 178.57,Z 602.24,A -85,B 0,C 180,E1 -22570.054,E2 -22570.054} C_VEL
LIN {X 0,Y 179.576,Z 605.077,A -85,B 0,C 180,E1 -22570.574,E2 -22570.574} C_VEL
LIN {X 0,Y 183.353,Z 613.674,A -85,B 0,C 180,E1 -22572.395,E2 -22572.395} C_VEL
LIN {X 0,Y 187.066,Z 624.236,A -85,B 0,C 180,E1 -22574.751,E2 -22574.751} C_VEL
LIN {X 0,Y 189.427,Z 632.633,A -85,B 0,C 180,E1 -22576.802,E2 -22576.802} C_VEL
LIN {X 0,Y 190.323,Z 637.472,A -85,B 0,C 180,E1 -22578.036,E2 -22578.036} C_VEL
LIN {X 0,Y 188.324,Z 647.251,A -85,B 0,C 180,E1 -22580.33,E2 -22580.33} C_VEL
LIN {X 0,Y 186.247,Z 656.256,A -85,B 0,C 180,E1 -22582.954,E2 -22582.954} C_VEL
LIN {X 0,Y 184.149,Z 665.053,A -85,B 0,C 180,E1 -22586.168,E2 -22586.168} C_VEL
LIN {X 0,Y 182.449,Z 671.992,A -85,B 0,C 180,E1 -22589.37,E2 -22589.37} C_VEL
LIN {X 0,Y 181.185,Z 676.973,A -85,B 0,C 180,E1 -22592.221,E2 -22592.221} C_VEL
LIN {X 0,Y 180.089,Z 681.677,A -85,B 0,C 180,E1 -22595.597,E2 -22595.597} C_VEL
LIN {X 0,Y 179.491,Z 685.272,A -85,B 0,C 180,E1 -22599.009,E2 -22599.009} C_VEL
LIN {X 0,Y 179.296,Z 687.232,A -85,B 0,C 180,E1 -22601.5,E2 -22601.5} C_VEL
LIN {X 0,Y 179.548,Z 689.516,A -85,B 0,C 180,E1 -22605.9,E2 -22605.9} C_VEL
LIN {X 0,Y 179.967,Z 690.118,A -85,B 0,C 180,E1 -22608.202,E2 -22608.202} C_VEL
LIN {X 0,Y 180.852,Z 690.263,A -85,B 0,C 180,E1 -22611.15,E2 -22611.15} C_VEL
LIN {X 0,Y 182.555,Z 689.437,A -85,B 0,C 180,E1 -22615.052,E2 -22615.052} C_VEL
LIN {X 0,Y 185.03,Z 687.173,A -85,B 0,C 180,E1 -22619.121,E2 -22619.121} C_VEL
LIN {X 0,Y 187.983,Z 683.738,A -85,B 0,C 180,E1 -22622.824,E2 -22622.824} C_VEL
LIN {X 0,Y 191.125,Z 679.485,A -85,B 0,C 180,E1 -22626.037,E2 -22626.037} C_VEL
LIN {X 0,Y 194.715,Z 673.959,A -85,B 0,C 180,E1 -22629.168,E2 -22629.168} C_VEL
LIN {X 0,Y 198.781,Z 666.898,A -85,B 0,C 180,E1 -22632.2,E2 -22632.2} C_VEL
LIN {X 0,Y 198.304,Z 665.567,A -85,B 0,C 180,E1 -22633.024,E2 -22633.024} C_VEL
LIN {X 0,Y 196.454,Z 664.092,A -85,B 0,C 180,E1 -22634.318,E2 -22634.318} C_VEL
LIN {X 0,Y 193.191,Z 662.185,A -85,B 0,C 180,E1 -22636.277,E2 -22636.277} C_VEL
LIN {X 0,Y 189.121,Z 661.361,A -85,B 0,C 180,E1 -22638.019,E2 -22638.019} C_VEL
LIN {X 0,Y 184.709,Z 661.178,A -85,B 0,C 180,E1 -22639.698,E2 -22639.698} C_VEL
LIN {X 0,Y 183.478,Z 660.506,A -85,B 0,C 180,E1 -22640.595,E2 -22640.595} C_VEL
LIN {X 0,Y 185.019,Z 672.373,A -85,B 0,C 180,E1 -22642.379,E2 -22642.379} C_VEL
LIN {X 0,Y 184.797,Z 676.151,A -85,B 0,C 180,E1 -22642.997,E2 -22642.997} C_VEL
LIN {X 0,Y 182.965,Z 687.865,A -85,B 0,C 180,E1 -22645.155,E2 -22645.155} C_VEL
LIN {X 0,Y 181.238,Z 698.832,A -85,B 0,C 180,E1 -22647.68,E2 -22647.68} C_VEL
LIN {X 0,Y 179.84,Z 707.561,A -85,B 0,C 180,E1 -22650.116,E2 -22650.116} C_VEL
LIN {X 0,Y 178.447,Z 716.311,A -85,B 0,C 180,E1 -22653.07,E2 -22653.07} C_VEL
LIN {X 0,Y 177.335,Z 724.888,A -85,B 0,C 180,E1 -22656.653,E2 -22656.653} C_VEL
LIN {X 0,Y 176.562,Z 731.795,A -85,B 0,C 180,E1 -22660.225,E2 -22660.225} C_VEL
LIN {X 0,Y 176.156,Z 737.311,A -85,B 0,C 180,E1 -22663.784,E2 -22663.784} C_VEL
LIN {X 0,Y 176.058,Z 741.592,A -85,B 0,C 180,E1 -22667.318,E2 -22667.318} C_VEL
LIN {X 0,Y 176.425,Z 744.819,A -85,B 0,C 180,E1 -22670.832,E2 -22670.832} C_VEL
LIN {X 0,Y 176.997,Z 746.451,A -85,B 0,C 180,E1 -22673.16,E2 -22673.16} C_VEL
LIN {X 0,Y 178.597,Z 748.538,A -85,B 0,C 180,E1 -22677.746,E2 -22677.746} C_VEL
LIN {X 0,Y 181.295,Z 749.159,A -85,B 0,C 180,E1 -22682.223,E2 -22682.223} C_VEL
LIN {X 0,Y 185.014,Z 748.268,A -85,B 0,C 180,E1 -22686.544,E2 -22686.544} C_VEL
LIN {X 0,Y 189.81,Z 745.987,A -85,B 0,C 180,E1 -22690.67,E2 -22690.67} C_VEL
LIN {X 0,Y 195.655,Z 742.117,A -85,B 0,C 180,E1 -22694.564,E2 -22694.564} C_VEL
LIN {X 0,Y 202.474,Z 736.684,A -85,B 0,C 180,E1 -22698.205,E2 -22698.205} C_VEL
LIN {X 0,Y 210.256,Z 729.303,A -85,B 0,C 180,E1 -22701.574,E2 -22701.574} C_VEL
LIN {X 0,Y 217.297,Z 721.607,A -85,B 0,C 180,E1 -22704.176,E2 -22704.176} C_VEL
LIN {X 0,Y 223.339,Z 714.087,A -85,B 0,C 180,E1 -22706.14,E2 -22706.14} C_VEL
LIN {X 0,Y 224.356,Z 712.419,A -85,B 0,C 180,E1 -22706.746,E2 -22706.746} C_VEL
LIN {X 0,Y 227.238,Z 706.162,A -85,B 0,C 180,E1 -22709.66,E2 -22709.66} C_VEL
LIN {X 0,Y 228.81,Z 702.65,A -85,B 0,C 180,E1 -22711.478,E2 -22711.478} C_VEL
LIN {X 0,Y 229.324,Z 701.271,A -85,B 0,C 180,E1 -22712.442,E2 -22712.442} C_VEL
LIN {X 0,Y 229.897,Z 699.483,A -85,B 0,C 180,E1 -22714.375,E2 -22714.375} C_VEL
LIN {X 0,Y 230.156,Z 698.787,A -85,B 0,C 180,E1 -22715.464,E2 -22715.464} C_VEL
LIN {X 0,Y 230.63,Z 698.099,A -85,B 0,C 180,E1 -22717.602,E2 -22717.602} C_VEL
LIN {X 0,Y 230.941,Z 698.512,A -85,B 0,C 180,E1 -22719.724,E2 -22719.724} C_VEL
LIN {X 0,Y 230.975,Z 698.895,A -85,B 0,C 180,E1 -22720.478,E2 -22720.478} C_VEL
LIN {X 0,Y 230.703,Z 700.709,A -85,B 0,C 180,E1 -22722.083,E2 -22722.083} C_VEL
LIN {X 0,Y 227.952,Z 706.976,A -85,B 0,C 180,E1 -22724.37,E2 -22724.37} C_VEL
LIN {X 0,Y 224.447,Z 714.323,A -85,B 0,C 180,E1 -22726.712,E2 -22726.712} C_VEL
LIN {X 0,Y 221.608,Z 719.59,A -85,B 0,C 180,E1 -22728.245,E2 -22728.245} C_VEL
LIN {X 0,Y 216.616,Z 726.965,A -85,B 0,C 180,E1 -22730.153,E2 -22730.153} C_VEL
LIN {X 0,Y 209.511,Z 736.191,A -85,B 0,C 180,E1 -22732.86,E2 -22732.86} C_VEL
LIN {X 0,Y 202.654,Z 743.975,A -85,B 0,C 180,E1 -22735.701,E2 -22735.701} C_VEL
LIN {X 0,Y 196.221,Z 750.454,A -85,B 0,C 180,E1 -22738.714,E2 -22738.714} C_VEL
LIN {X 0,Y 189.991,Z 756.222,A -85,B 0,C 180,E1 -22742.461,E2 -22742.461} C_VEL
LIN {X 0,Y 185.998,Z 759.596,A -85,B 0,C 180,E1 -22745.443,E2 -22745.443} C_VEL
LIN {X 0,Y 181.84,Z 762.839,A -85,B 0,C 180,E1 -22749.647,E2 -22749.647} C_VEL
LIN {X 0,Y 178.715,Z 764.75,A -85,B 0,C 180,E1 -22754.024,E2 -22754.024} C_VEL
LIN {X 0,Y 177.058,Z 765.279,A -85,B 0,C 180,E1 -22758.555,E2 -22758.555} C_VEL
LIN {X 0,Y 176.488,Z 764.415,A -85,B 0,C 180,E1 -22763.141,E2 -22763.141} C_VEL
LIN {X 0,Y 176.547,Z 763.817,A -85,B 0,C 180,E1 -22764.694,E2 -22764.694} C_VEL
LIN {X 0,Y 175.949,Z 762.739,A -85,B 0,C 180,E1 -22766.568,E2 -22766.568} C_VEL
LIN {X 0,Y 174.483,Z 761.237,A -85,B 0,C 180,E1 -22768.388,E2 -22768.388} C_VEL
LIN {X 0,Y 171.027,Z 757.228,A -85,B 0,C 180,E1 -22771.987,E2 -22771.987} C_VEL
LIN {X 0,Y 170.082,Z 754.852,A -85,B 0,C 180,E1 -22773.829,E2 -22773.829} C_VEL
LIN {X 0,Y 170.019,Z 754.007,A -85,B 0,C 180,E1 -22774.45,E2 -22774.45} C_VEL
LIN {X 0,Y 170.088,Z 749.628,A -85,B 0,C 180,E1 -22777.391,E2 -22777.391} C_VEL
LIN {X 0,Y 170.515,Z 742.312,A -85,B 0,C 180,E1 -22781.292,E2 -22781.292} C_VEL
LIN {X 0,Y 171.445,Z 733.925,A -85,B 0,C 180,E1 -22784.847,E2 -22784.847} C_VEL
LIN {X 0,Y 172.638,Z 725.418,A -85,B 0,C 180,E1 -22787.78,E2 -22787.78} C_VEL
LIN {X 0,Y 174.302,Z 714.993,A -85,B 0,C 180,E1 -22790.661,E2 -22790.661} C_VEL
LIN {X 0,Y 175.224,Z 708.85,A -85,B 0,C 180,E1 -22792.097,E2 -22792.097} C_VEL
LIN {X 0,Y 175.353,Z 703.848,A -85,B 0,C 180,E1 -22793.206,E2 -22793.206} C_VEL
LIN {X 0,Y 175.953,Z 693.114,A -85,B 0,C 180,E1 -22796.385,E2 -22796.385} C_VEL
LIN {X 0,Y 176.624,Z 681.784,A -85,B 0,C 180,E1 -22799.109,E2 -22799.109} C_VEL
LIN {X 0,Y 176.97,Z 670.353,A -85,B 0,C 180,E1 -22801.337,E2 -22801.337} C_VEL
LIN {X 0,Y 176.793,Z 657.29,A -85,B 0,C 180,E1 -22803.403,E2 -22803.403} C_VEL
LIN {X 0,Y 176,Z 644.067,A -85,B 0,C 180,E1 -22805.074,E2 -22805.074} C_VEL
LIN {X 0,Y 174.237,Z 630.554,A -85,B 0,C 180,E1 -22806.428,E2 -22806.428} C_VEL
LIN {X 0,Y 174.075,Z 628.812,A -85,B 0,C 180,E1 -22806.561,E2 -22806.561} C_VEL
LIN {X 0,Y 175.316,Z 624.223,A -85,B 0,C 180,E1 -22809.899,E2 -22809.899} C_VEL
LIN {X 0,Y 175.129,Z 621.571,A -85,B 0,C 180,E1 -22811.938,E2 -22811.938} C_VEL
LIN {X 0,Y 173.832,Z 615.657,A -85,B 0,C 180,E1 -22816.7,E2 -22816.7} C_VEL
LIN {X 0,Y 172.696,Z 609.177,A -85,B 0,C 180,E1 -22822.378,E2 -22822.378} C_VEL
LIN {X 0,Y 171.527,Z 603.495,A -85,B 0,C 180,E1 -22827.814,E2 -22827.814} C_VEL
LIN {X 0,Y 171.471,Z 603.131,A -85,B 0,C 180,E1 -22828.262,E2 -22828.262} C_VEL
LIN {X 0,Y 171.426,Z 603.131,A -85,B 0,C 180,E1 -22833.193,E2 -22833.193} C_VEL
LIN {X 0,Y 171.469,Z 603.128,A -85,B 0,C 180,E1 -22838.352,E2 -22838.352} C_VEL
LIN {X 0,Y 171.586,Z 603.113,A -85,B 0,C 180,E1 -22840.871,E2 -22840.871} C_VEL
LIN {X 0,Y 171.616,Z 603.111,A -85,B 0,C 180,E1 -22845.775,E2 -22845.775} C_VEL
LIN {X 0,Y 171.917,Z 603.071,A -85,B 0,C 180,E1 -22850.588,E2 -22850.588} C_VEL
LIN {X 0,Y 171.83,Z 603.08,A -85,B 0,C 180,E1 -22855.307,E2 -22855.307} C_VEL
LIN {X 0,Y 172.339,Z 603.018,A -85,B 0,C 180,E1 -22859.999,E2 -22859.999} C_VEL
LIN {X 0,Y 171.825,Z 603.058,A -85,B 0,C 180,E1 -22864.691,E2 -22864.691} C_VEL
LIN {X 0,Y 171.894,Z 603.071,A -85,B 0,C 180,E1 -22869.412,E2 -22869.412} C_VEL
LIN {X 0,Y 171.598,Z 603.095,A -85,B 0,C 180,E1 -22874.224,E2 -22874.224} C_VEL
LIN {X 0,Y 171.549,Z 603.112,A -85,B 0,C 180,E1 -22879.56,E2 -22879.56} C_VEL
LIN {X 0,Y 171.473,Z 603.11,A -85,B 0,C 180,E1 -22885.615,E2 -22885.615} C_VEL
LIN {X 0,Y 171.462,Z 603.126,A -85,B 0,C 180,E1 -22890.594,E2 -22890.594} C_VEL
LIN {X 0,Y 171.396,Z 603.134,A -85,B 0,C 180,E1 -22895.033,E2 -22895.033} C_VEL
LIN {X 0,Y 171.36,Z 603.136,A -85,B 0,C 180,E1 -22898.806,E2 -22898.806} C_VEL
LIN {X 0,Y 171.345,Z 603.127,A -85,B 0,C 180,E1 -22904.208,E2 -22904.208} C_VEL
LIN {X 0,Y 171.363,Z 603.137,A -85,B 0,C 180,E1 -22908.987,E2 -22908.987} C_VEL
LIN {X 0,Y 171.418,Z 603.12,A -85,B 0,C 180,E1 -22912.047,E2 -22912.047} C_VEL
LIN {X 0,Y 171.412,Z 603.133,A -85,B 0,C 180,E1 -22915.084,E2 -22915.084} C_VEL
LIN {X 0,Y 171.449,Z 603.129,A -85,B 0,C 180,E1 -22920.532,E2 -22920.532} C_VEL
LIN {X 0,Y 171.458,Z 603.128,A -85,B 0,C 180,E1 -22925.8,E2 -22925.8} C_VEL
LIN {X 0,Y 171.497,Z 603.226,A -85,B 0,C 180,E1 -22928.773,E2 -22928.773} C_VEL
LIN {X 0,Y 172.712,Z 606.282,A -85,B 0,C 180,E1 -22929.374,E2 -22929.374} C_VEL
LIN {X 0,Y 176.724,Z 615.492,A -85,B 0,C 180,E1 -22931.447,E2 -22931.447} C_VEL
LIN {X 0,Y 179.915,Z 624.154,A -85,B 0,C 180,E1 -22933.522,E2 -22933.522} C_VEL
LIN {X 0,Y 182.623,Z 633.706,A -85,B 0,C 180,E1 -22935.954,E2 -22935.954} C_VEL
LIN {X 0,Y 183.7,Z 638.61,A -85,B 0,C 180,E1 -22937.29,E2 -22937.29} C_VEL
LIN {X 0,Y 181.856,Z 647.464,A -85,B 0,C 180,E1 -22939.42,E2 -22939.42} C_VEL
LIN {X 0,Y 179.667,Z 656.609,A -85,B 0,C 180,E1 -22942.129,E2 -22942.129} C_VEL
LIN {X 0,Y 177.425,Z 665.519,A -85,B 0,C 180,E1 -22945.454,E2 -22945.454} C_VEL
LIN {X 0,Y 175.758,Z 672.023,A -85,B 0,C 180,E1 -22948.494,E2 -22948.494} C_VEL
LIN {X 0,Y 174.055,Z 678.51,A -85,B 0,C 180,E1 -22952.312,E2 -22952.312} C_VEL
LIN {X 0,Y 172.977,Z 683.088,A -85,B 0,C 180,E1 -22955.828,E2 -22955.828} C_VEL
LIN {X 0,Y 172.397,Z 686.586,A -85,B 0,C 180,E1 -22959.383,E2 -22959.383} C_VEL
LIN {X 0,Y 172.244,Z 688.347,A -85,B 0,C 180,E1 -22961.769,E2 -22961.769} C_VEL
LIN {X 0,Y 172.319,Z 689.705,A -85,B 0,C 180,E1 -22964.162,E2 -22964.162} C_VEL
LIN {X 0,Y 172.614,Z 690.662,A -85,B 0,C 180,E1 -22966.557,E2 -22966.557} C_VEL
LIN {X 0,Y 173.104,Z 691.177,A -85,B 0,C 180,E1 -22968.951,E2 -22968.951} C_VEL
LIN {X 0,Y 173.994,Z 691.284,A -85,B 0,C 180,E1 -22971.72,E2 -22971.72} C_VEL
LIN {X 0,Y 175.991,Z 690.325,A -85,B 0,C 180,E1 -22976.055,E2 -22976.055} C_VEL
LIN {X 0,Y 178.5,Z 688.148,A -85,B 0,C 180,E1 -22979.982,E2 -22979.982} C_VEL
LIN {X 0,Y 181.894,Z 684.405,A -85,B 0,C 180,E1 -22984.07,E2 -22984.07} C_VEL
LIN {X 0,Y 185.268,Z 680.039,A -85,B 0,C 180,E1 -22987.366,E2 -22987.366} C_VEL
LIN {X 0,Y 189.116,Z 674.367,A -85,B 0,C 180,E1 -22990.564,E2 -22990.564} C_VEL
LIN {X 0,Y 191.592,Z 670.258,A -85,B 0,C 180,E1 -22992.422,E2 -22992.422} C_VEL
LIN {X 0,Y 192.073,Z 669.105,A -85,B 0,C 180,E1 -22992.963,E2 -22992.963} C_VEL
LIN {X 0,Y 188.973,Z 667.164,A -85,B 0,C 180,E1 -22995.041,E2 -22995.041} C_VEL
LIN {X 0,Y 185.17,Z 666.14,A -85,B 0,C 180,E1 -22996.909,E2 -22996.909} C_VEL
LIN {X 0,Y 180.735,Z 665.965,A -85,B 0,C 180,E1 -22998.621,E2 -22998.621} C_VEL
LIN {X 0,Y 177.108,Z 665.053,A -85,B 0,C 180,E1 -23000.588,E2 -23000.588} C_VEL
LIN {X 0,Y 176.992,Z 664.828,A -85,B 0,C 180,E1 -23000.759,E2 -23000.759} C_VEL
LIN {X 0,Y 178.016,Z 673.224,A -85,B 0,C 180,E1 -23002.143,E2 -23002.143} C_VEL
LIN {X 0,Y 176.787,Z 682.33,A -85,B 0,C 180,E1 -23003.749,E2 -23003.749} C_VEL
LIN {X 0,Y 174.778,Z 694.906,A -85,B 0,C 180,E1 -23006.504,E2 -23006.504} C_VEL
LIN {X 0,Y 173.009,Z 705.768,A -85,B 0,C 180,E1 -23009.485,E2 -23009.485} C_VEL
LIN {X 0,Y 171.3,Z 716.513,A -85,B 0,C 180,E1 -23013.174,E2 -23013.174} C_VEL
LIN {X 0,Y 170.182,Z 725.136,A -85,B 0,C 180,E1 -23016.902,E2 -23016.902} C_VEL
LIN {X 0,Y 169.415,Z 732.069,A -85,B 0,C 180,E1 -23020.619,E2 -23020.619} C_VEL
LIN {X 0,Y 169.022,Z 737.554,A -85,B 0,C 180,E1 -23024.321,E2 -23024.321} C_VEL
LIN {X 0,Y 168.996,Z 741.862,A -85,B 0,C 180,E1 -23028,E2 -23028} C_VEL
LIN {X 0,Y 169.26,Z 744.164,A -85,B 0,C 180,E1 -23030.441,E2 -23030.441} C_VEL
LIN {X 0,Y 169.882,Z 746.215,A -85,B 0,C 180,E1 -23033.134,E2 -23033.134} C_VEL
LIN {X 0,Y 171.38,Z 748.596,A -85,B 0,C 180,E1 -23037.651,E2 -23037.651} C_VEL
LIN {X 0,Y 174.089,Z 749.655,A -85,B 0,C 180,E1 -23042.315,E2 -23042.315} C_VEL
LIN {X 0,Y 177.9,Z 749.277,A -85,B 0,C 180,E1 -23046.807,E2 -23046.807} C_VEL
LIN {X 0,Y 182.823,Z 747.473,A -85,B 0,C 180,E1 -23051.083,E2 -23051.083} C_VEL
LIN {X 0,Y 188.828,Z 744.181,A -85,B 0,C 180,E1 -23055.103,E2 -23055.103} C_VEL
LIN {X 0,Y 193.994,Z 740.678,A -85,B 0,C 180,E1 -23057.936,E2 -23057.936} C_VEL
LIN {X 0,Y 199.729,Z 736.232,A -85,B 0,C 180,E1 -23060.603,E2 -23060.603} C_VEL
LIN {X 0,Y 206.768,Z 729.956,A -85,B 0,C 180,E1 -23063.41,E2 -23063.41} C_VEL
LIN {X 0,Y 213.788,Z 722.837,A -85,B 0,C 180,E1 -23065.823,E2 -23065.823} C_VEL
LIN {X 0,Y 218.511,Z 717.449,A -85,B 0,C 180,E1 -23067.28,E2 -23067.28} C_VEL
LIN {X 0,Y 219.453,Z 716.233,A -85,B 0,C 180,E1 -23067.67,E2 -23067.67} C_VEL
LIN {X 0,Y 222.567,Z 710.819,A -85,B 0,C 180,E1 -23070.348,E2 -23070.348} C_VEL
LIN {X 0,Y 224.472,Z 707.339,A -85,B 0,C 180,E1 -23072.295,E2 -23072.295} C_VEL
LIN {X 0,Y 225.434,Z 705.396,A -85,B 0,C 180,E1 -23074.137,E2 -23074.137} C_VEL
LIN {X 0,Y 226.031,Z 704.243,A -85,B 0,C 180,E1 -23076.212,E2 -23076.212} C_VEL
LIN {X 0,Y 226.482,Z 703.955,A -85,B 0,C 180,E1 -23078.363,E2 -23078.363} C_VEL
LIN {X 0,Y 226.629,Z 704.106,A -85,B 0,C 180,E1 -23079.173,E2 -23079.173} C_VEL
LIN {X 0,Y 226.581,Z 704.939,A -85,B 0,C 180,E1 -23080.646,E2 -23080.646} C_VEL
LIN {X 0,Y 225.975,Z 706.613,A -85,B 0,C 180,E1 -23081.722,E2 -23081.722} C_VEL
LIN {X 0,Y 222.695,Z 712.723,A -85,B 0,C 180,E1 -23083.972,E2 -23083.972} C_VEL
LIN {X 0,Y 218.413,Z 720.032,A -85,B 0,C 180,E1 -23086.358,E2 -23086.358} C_VEL
LIN {X 0,Y 214.741,Z 725.369,A -85,B 0,C 180,E1 -23087.865,E2 -23087.865} C_VEL
LIN {X 0,Y 207.189,Z 734.592,A -85,B 0,C 180,E1 -23090.508,E2 -23090.508} C_VEL
LIN {X 0,Y 200.023,Z 742.424,A -85,B 0,C 180,E1 -23093.325,E2 -23093.325} C_VEL
LIN {X 0,Y 192.048,Z 749.849,A -85,B 0,C 180,E1 -23096.709,E2 -23096.709} C_VEL
LIN {X 0,Y 185.334,Z 755.593,A -85,B 0,C 180,E1 -23100.467,E2 -23100.467} C_VEL
LIN {X 0,Y 181.566,Z 758.421,A -85,B 0,C 180,E1 -23102.91,E2 -23102.91} C_VEL
LIN {X 0,Y 177.256,Z 761.539,A -85,B 0,C 180,E1 -23106.644,E2 -23106.644} C_VEL
LIN {X 0,Y 173.393,Z 763.771,A -85,B 0,C 180,E1 -23111.082,E2 -23111.082} C_VEL
LIN {X 0,Y 170.833,Z 764.689,A -85,B 0,C 180,E1 -23115.712,E2 -23115.712} C_VEL
LIN {X 0,Y 169.639,Z 764.291,A -85,B 0,C 180,E1 -23120.463,E2 -23120.463} C_VEL
LIN {X 0,Y 169.563,Z 762.472,A -85,B 0,C 180,E1 -23125.247,E2 -23125.247} C_VEL
LIN {X 0,Y 169.773,Z 760.983,A -85,B 0,C 180,E1 -23127.63,E2 -23127.63} C_VEL
LIN {X 0,Y 170.157,Z 759.098,A -85,B 0,C 180,E1 -23130.002,E2 -23130.002} C_VEL
LIN {X 0,Y 170.019,Z 755.18,A -85,B 0,C 180,E1 -23133.557,E2 -23133.557} C_VEL
LIN {X 0,Y 170.019,Z 754.007,A -85,B 0,C 180,E1 -23134.45,E2 -23134.45} C_VEL
LIN {X 0,Y 169.74,Z 752.304,A -85,B 0,C 180,E1 -23135.641,E2 -23135.641} C_VEL
LIN {X 0,Y 168.476,Z 749.435,A -85,B 0,C 180,E1 -23137.343,E2 -23137.343} C_VEL
LIN {X 0,Y 164.597,Z 741.696,A -85,B 0,C 180,E1 -23141.124,E2 -23141.124} C_VEL
LIN {X 0,Y 163.914,Z 738.039,A -85,B 0,C 180,E1 -23142.757,E2 -23142.757} C_VEL
LIN {X 0,Y 163.985,Z 736.781,A -85,B 0,C 180,E1 -23143.302,E2 -23143.302} C_VEL
LIN {X 0,Y 165.13,Z 728.011,A -85,B 0,C 180,E1 -23146.698,E2 -23146.698} C_VEL
LIN {X 0,Y 166.783,Z 717.299,A -85,B 0,C 180,E1 -23150.024,E2 -23150.024} C_VEL
LIN {X 0,Y 168.178,Z 707.628,A -85,B 0,C 180,E1 -23152.45,E2 -23152.45} C_VEL
LIN {X 0,Y 168.239,Z 705.514,A -85,B 0,C 180,E1 -23152.986,E2 -23152.986} C_VEL
LIN {X 0,Y 168.873,Z 695.623,A -85,B 0,C 180,E1 -23156.245,E2 -23156.245} C_VEL
LIN {X 0,Y 169.613,Z 684.871,A -85,B 0,C 180,E1 -23159.128,E2 -23159.128} C_VEL
LIN {X 0,Y 170.184,Z 674.397,A -85,B 0,C 180,E1 -23161.426,E2 -23161.426} C_VEL
LIN {X 0,Y 170.324,Z 661.808,A -85,B 0,C 180,E1 -23163.699,E2 -23163.699} C_VEL
LIN {X 0,Y 169.906,Z 648.822,A -85,B 0,C 180,E1 -23165.591,E2 -23165.591} C_VEL
LIN {X 0,Y 168.576,Z 635.071,A -85,B 0,C 180,E1 -23167.186,E2 -23167.186} C_VEL
LIN {X 0,Y 167.508,Z 627.727,A -85,B 0,C 180,E1 -23167.963,E2 -23167.963} C_VEL
LIN {X 0,Y 168.235,Z 625.048,A -85,B 0,C 180,E1 -23169.997,E2 -23169.997} C_VEL
LIN {X 0,Y 168.093,Z 622.557,A -85,B 0,C 180,E1 -23171.99,E2 -23171.99} C_VEL
LIN {X 0,Y 166.68,Z 615.987,A -85,B 0,C 180,E1 -23177.573,E2 -23177.573} C_VEL
LIN {X 0,Y 165.818,Z 611.002,A -85,B 0,C 180,E1 -23182.079,E2 -23182.079} C_VEL
LIN {X 0,Y 164.684,Z 605.361,A -85,B 0,C 180,E1 -23187.68,E2 -23187.68} C_VEL
LIN {X 0,Y 164.409,Z 604.009,A -85,B 0,C 180,E1 -23189.137,E2 -23189.137} C_VEL
LIN {X 0,Y 164.423,Z 604.005,A -85,B 0,C 180,E1 -23194.694,E2 -23194.694} C_VEL
LIN {X 0,Y 164.491,Z 603.998,A -85,B 0,C 180,E1 -23200.051,E2 -23200.051} C_VEL
LIN {X 0,Y 164.56,Z 603.99,A -85,B 0,C 180,E1 -23205.152,E2 -23205.152} C_VEL
LIN {X 0,Y 164.859,Z 603.953,A -85,B 0,C 180,E1 -23210.181,E2 -23210.181} C_VEL
LIN {X 0,Y 164.868,Z 603.948,A -85,B 0,C 180,E1 -23212.652,E2 -23212.652} C_VEL
LIN {X 0,Y 165.301,Z 603.895,A -85,B 0,C 180,E1 -23219.999,E2 -23219.999} C_VEL
LIN {X 0,Y 164.835,Z 603.94,A -85,B 0,C 180,E1 -23227.113,E2 -23227.113} C_VEL
LIN {X 0,Y 164.759,Z 603.96,A -85,B 0,C 180,E1 -23231.15,E2 -23231.15} C_VEL
LIN {X 0,Y 164.489,Z 603.978,A -85,B 0,C 180,E1 -23237.402,E2 -23237.402} C_VEL
LIN {X 0,Y 164.478,Z 603.993,A -85,B 0,C 180,E1 -23239.987,E2 -23239.987} C_VEL
LIN {X 0,Y 164.398,Z 603.987,A -85,B 0,C 180,E1 -23246.132,E2 -23246.132} C_VEL
LIN {X 0,Y 164.392,Z 604.007,A -85,B 0,C 180,E1 -23251.234,E2 -23251.234} C_VEL
LIN {X 0,Y 164.297,Z 604.019,A -85,B 0,C 180,E1 -23256.787,E2 -23256.787} C_VEL
LIN {X 0,Y 164.295,Z 604.017,A -85,B 0,C 180,E1 -23259.914,E2 -23259.914} C_VEL
LIN {X 0,Y 164.282,Z 604.013,A -85,B 0,C 180,E1 -23263.34,E2 -23263.34} C_VEL
LIN {X 0,Y 164.294,Z 604.011,A -85,B 0,C 180,E1 -23266.807,E2 -23266.807} C_VEL
LIN {X 0,Y 164.312,Z 604.011,A -85,B 0,C 180,E1 -23270.343,E2 -23270.343} C_VEL
LIN {X 0,Y 164.345,Z 604.01,A -85,B 0,C 180,E1 -23274.34,E2 -23274.34} C_VEL
LIN {X 0,Y 164.39,Z 604.001,A -85,B 0,C 180,E1 -23279.132,E2 -23279.132} C_VEL
LIN {X 0,Y 164.417,Z 604.003,A -85,B 0,C 180,E1 -23284.692,E2 -23284.692} C_VEL
LIN {X 0,Y 164.389,Z 604.105,A -85,B 0,C 180,E1 -23287.327,E2 -23287.327} C_VEL
LIN {X 0,Y 165.242,Z 606.574,A -85,B 0,C 180,E1 -23287.817,E2 -23287.817} C_VEL
LIN {X 0,Y 170.02,Z 616.692,A -85,B 0,C 180,E1 -23290.311,E2 -23290.311} C_VEL
LIN {X 0,Y 173.492,Z 626.475,A -85,B 0,C 180,E1 -23292.781,E2 -23292.781} C_VEL
LIN {X 0,Y 176.278,Z 636.609,A -85,B 0,C 180,E1 -23295.562,E2 -23295.562} C_VEL
LIN {X 0,Y 176.974,Z 639.891,A -85,B 0,C 180,E1 -23296.506,E2 -23296.506} C_VEL
LIN {X 0,Y 175.446,Z 647.609,A -85,B 0,C 180,E1 -23298.444,E2 -23298.444} C_VEL
LIN {X 0,Y 173.101,Z 656.957,A -85,B 0,C 180,E1 -23301.24,E2 -23301.24} C_VEL
LIN {X 0,Y 170.734,Z 665.974,A -85,B 0,C 180,E1 -23304.684,E2 -23304.684} C_VEL
LIN {X 0,Y 168.746,Z 673.392,A -85,B 0,C 180,E1 -23308.269,E2 -23308.269} C_VEL
LIN {X 0,Y 166.937,Z 680.007,A -85,B 0,C 180,E1 -23312.411,E2 -23312.411} C_VEL
LIN {X 0,Y 165.879,Z 684.477,A -85,B 0,C 180,E1 -23316.078,E2 -23316.078} C_VEL
LIN {X 0,Y 165.318,Z 687.879,A -85,B 0,C 180,E1 -23319.788,E2 -23319.788} C_VEL
LIN {X 0,Y 165.226,Z 689.59,A -85,B 0,C 180,E1 -23322.277,E2 -23322.277} C_VEL
LIN {X 0,Y 165.346,Z 690.904,A -85,B 0,C 180,E1 -23324.773,E2 -23324.773} C_VEL
LIN {X 0,Y 165.686,Z 691.775,A -85,B 0,C 180,E1 -23327.27,E2 -23327.27} C_VEL
LIN {X 0,Y 167.13,Z 692.306,A -85,B 0,C 180,E1 -23332.236,E2 -23332.236} C_VEL
LIN {X 0,Y 168.174,Z 691.98,A -85,B 0,C 180,E1 -23334.699,E2 -23334.699} C_VEL
LIN {X 0,Y 169.468,Z 691.197,A -85,B 0,C 180,E1 -23337.138,E2 -23337.138} C_VEL
LIN {X 0,Y 172.036,Z 689.112,A -85,B 0,C 180,E1 -23340.921,E2 -23340.921} C_VEL
LIN {X 0,Y 174.804,Z 686.28,A -85,B 0,C 180,E1 -23344.252,E2 -23344.252} C_VEL
LIN {X 0,Y 178.818,Z 681.453,A -85,B 0,C 180,E1 -23348.184,E2 -23348.184} C_VEL
LIN {X 0,Y 182.906,Z 675.827,A -85,B 0,C 180,E1 -23351.512,E2 -23351.512} C_VEL
LIN {X 0,Y 185.06,Z 672.49,A -85,B 0,C 180,E1 -23353.121,E2 -23353.121} C_VEL
LIN {X 0,Y 184.565,Z 671.9,A -85,B 0,C 180,E1 -23353.658,E2 -23353.658} C_VEL
LIN {X 0,Y 181.038,Z 670.702,A -85,B 0,C 180,E1 -23355.673,E2 -23355.673} C_VEL
LIN {X 0,Y 176.657,Z 670.462,A -85,B 0,C 180,E1 -23357.445,E2 -23357.445} C_VEL
LIN {X 0,Y 170.825,Z 669.445,A -85,B 0,C 180,E1 -23360.526,E2 -23360.526} C_VEL
LIN {X 0,Y 170.413,Z 669.052,A -85,B 0,C 180,E1 -23361.075,E2 -23361.075} C_VEL
LIN {X 0,Y 170.965,Z 673.965,A -85,B 0,C 180,E1 -23361.932,E2 -23361.932} C_VEL
LIN {X 0,Y 169.027,Z 686.797,A -85,B 0,C 180,E1 -23364.402,E2 -23364.402} C_VEL
LIN {X 0,Y 167.136,Z 698.417,A -85,B 0,C 180,E1 -23367.24,E2 -23367.24} C_VEL
LIN {X 0,Y 165.533,Z 707.863,A -85,B 0,C 180,E1 -23370.076,E2 -23370.076} C_VEL
LIN {X 0,Y 164.12,Z 716.987,A -85,B 0,C 180,E1 -23373.395,E2 -23373.395} C_VEL
LIN {X 0,Y 163.016,Z 725.308,A -85,B 0,C 180,E1 -23377.17,E2 -23377.17} C_VEL
LIN {X 0,Y 162.297,Z 732.222,A -85,B 0,C 180,E1 -23381.049,E2 -23381.049} C_VEL
LIN {X 0,Y 161.932,Z 737.763,A -85,B 0,C 180,E1 -23384.907,E2 -23384.907} C_VEL
LIN {X 0,Y 161.967,Z 742.126,A -85,B 0,C 180,E1 -23388.741,E2 -23388.741} C_VEL
LIN {X 0,Y 162.778,Z 745.949,A -85,B 0,C 180,E1 -23393.209,E2 -23393.209} C_VEL
LIN {X 0,Y 164.174,Z 748.487,A -85,B 0,C 180,E1 -23397.547,E2 -23397.547} C_VEL
LIN {X 0,Y 166.907,Z 750.01,A -85,B 0,C 180,E1 -23402.414,E2 -23402.414} C_VEL
LIN {X 0,Y 170.772,Z 750.138,A -85,B 0,C 180,E1 -23407.093,E2 -23407.093} C_VEL
LIN {X 0,Y 175.827,Z 748.817,A -85,B 0,C 180,E1 -23411.529,E2 -23411.529} C_VEL
LIN {X 0,Y 182.008,Z 746.066,A -85,B 0,C 180,E1 -23415.683,E2 -23415.683} C_VEL
LIN {X 0,Y 189.204,Z 741.828,A -85,B 0,C 180,E1 -23419.531,E2 -23419.531} C_VEL
LIN {X 0,Y 195.271,Z 737.53,A -85,B 0,C 180,E1 -23422.205,E2 -23422.205} C_VEL
LIN {X 0,Y 204.132,Z 730.219,A -85,B 0,C 180,E1 -23425.491,E2 -23425.491} C_VEL
LIN {X 0,Y 211.271,Z 723.329,A -85,B 0,C 180,E1 -23427.757,E2 -23427.757} C_VEL
LIN {X 0,Y 214.89,Z 719.47,A -85,B 0,C 180,E1 -23428.843,E2 -23428.843} C_VEL
LIN {X 0,Y 218.912,Z 713.653,A -85,B 0,C 180,E1 -23432.02,E2 -23432.02} C_VEL
LIN {X 0,Y 219.901,Z 712.221,A -85,B 0,C 180,E1 -23432.911,E2 -23432.911} C_VEL
LIN {X 0,Y 220.997,Z 710.409,A -85,B 0,C 180,E1 -23434.92,E2 -23434.92} C_VEL
LIN {X 0,Y 221.774,Z 709.533,A -85,B 0,C 180,E1 -23437.607,E2 -23437.607} C_VEL
LIN {X 0,Y 222.132,Z 709.703,A -85,B 0,C 180,E1 -23439.256,E2 -23439.256} C_VEL
LIN {X 0,Y 221.857,Z 710.648,A -85,B 0,C 180,E1 -23440.515,E2 -23440.515} C_VEL
LIN {X 0,Y 220.413,Z 713.131,A -85,B 0,C 180,E1 -23441.642,E2 -23441.642} C_VEL
LIN {X 0,Y 216.451,Z 719.19,A -85,B 0,C 180,E1 -23443.884,E2 -23443.884} C_VEL
LIN {X 0,Y 213.039,Z 724.096,A -85,B 0,C 180,E1 -23445.494,E2 -23445.494} C_VEL
LIN {X 0,Y 207.552,Z 730.633,A -85,B 0,C 180,E1 -23447.376,E2 -23447.376} C_VEL
LIN {X 0,Y 199.791,Z 738.908,A -85,B 0,C 180,E1 -23450.064,E2 -23450.064} C_VEL
LIN {X 0,Y 192.349,Z 745.88,A -85,B 0,C 180,E1 -23452.927,E2 -23452.927} C_VEL
LIN {X 0,Y 186.225,Z 750.915,A -85,B 0,C 180,E1 -23455.525,E2 -23455.525} C_VEL
LIN {X 0,Y 179.227,Z 756.232,A -85,B 0,C 180,E1 -23459.354,E2 -23459.354} C_VEL
LIN {X 0,Y 175.024,Z 758.98,A -85,B 0,C 180,E1 -23462.057,E2 -23462.057} C_VEL
LIN {X 0,Y 170.759,Z 761.58,A -85,B 0,C 180,E1 -23465.699,E2 -23465.699} C_VEL
LIN {X 0,Y 166.683,Z 763.532,A -85,B 0,C 180,E1 -23470.289,E2 -23470.289} C_VEL
LIN {X 0,Y 163.943,Z 764.173,A -85,B 0,C 180,E1 -23475.098,E2 -23475.098} C_VEL
LIN {X 0,Y 162.648,Z 763.464,A -85,B 0,C 180,E1 -23480.049,E2 -23480.049} C_VEL
LIN {X 0,Y 162.56,Z 761.404,A -85,B 0,C 180,E1 -23485.042,E2 -23485.042} C_VEL
LIN {X 0,Y 162.947,Z 758.823,A -85,B 0,C 180,E1 -23488.767,E2 -23488.767} C_VEL
LIN {X 0,Y 163.148,Z 757.777,A -85,B 0,C 180,E1 -23490.002,E2 -23490.002} C_VEL
LIN {X 0,Y 163.023,Z 752.921,A -85,B 0,C 180,E1 -23494.273,E2 -23494.273} C_VEL
LIN {X 0,Y 163.097,Z 747.922,A -85,B 0,C 180,E1 -23497.646,E2 -23497.646} C_VEL
LIN {X 0,Y 163.609,Z 740.175,A -85,B 0,C 180,E1 -23501.776,E2 -23501.776} C_VEL
LIN {X 0,Y 163.985,Z 736.781,A -85,B 0,C 180,E1 -23503.302,E2 -23503.302} C_VEL
LIN {X 0,Y 163.81,Z 732.928,A -85,B 0,C 180,E1 -23504.866,E2 -23504.866} C_VEL
LIN {X 0,Y 161.833,Z 726.022,A -85,B 0,C 180,E1 -23507.277,E2 -23507.277} C_VEL
LIN {X 0,Y 160.036,Z 718.613,A -85,B 0,C 180,E1 -23509.562,E2 -23509.562} C_VEL
LIN {X 0,Y 160.165,Z 713.944,A -85,B 0,C 180,E1 -23510.878,E2 -23510.878} C_VEL
LIN {X 0,Y 161.098,Z 707.376,A -85,B 0,C 180,E1 -23512.612,E2 -23512.612} C_VEL
LIN {X 0,Y 161.729,Z 697.864,A -85,B 0,C 180,E1 -23516.105,E2 -23516.105} C_VEL
LIN {X 0,Y 162.636,Z 687.269,A -85,B 0,C 180,E1 -23519.244,E2 -23519.244} C_VEL
LIN {X 0,Y 163.458,Z 675.214,A -85,B 0,C 180,E1 -23522.148,E2 -23522.148} C_VEL
LIN {X 0,Y 163.759,Z 662.927,A -85,B 0,C 180,E1 -23524.545,E2 -23524.545} C_VEL
LIN {X 0,Y 163.534,Z 650.128,A -85,B 0,C 180,E1 -23526.557,E2 -23526.557} C_VEL
LIN {X 0,Y 162.429,Z 636.521,A -85,B 0,C 180,E1 -23528.305,E2 -23528.305} C_VEL
LIN {X 0,Y 160.925,Z 626.749,A -85,B 0,C 180,E1 -23529.376,E2 -23529.376} C_VEL
LIN {X 0,Y 161.178,Z 624.939,A -85,B 0,C 180,E1 -23530.851,E2 -23530.851} C_VEL
LIN {X 0,Y 160.662,Z 621.924,A -85,B 0,C 180,E1 -23533.442,E2 -23533.442} C_VEL
LIN {X 0,Y 159.488,Z 616.162,A -85,B 0,C 180,E1 -23538.623,E2 -23538.623} C_VEL
LIN {X 0,Y 158.748,Z 611.724,A -85,B 0,C 180,E1 -23542.837,E2 -23542.837} C_VEL
LIN {X 0,Y 157.766,Z 606.95,A -85,B 0,C 180,E1 -23547.825,E2 -23547.825} C_VEL
LIN {X 0,Y 157.309,Z 604.892,A -85,B 0,C 180,E1 -23550.195,E2 -23550.195} C_VEL
LIN {X 0,Y 157.329,Z 604.887,A -85,B 0,C 180,E1 -23553.466,E2 -23553.466} C_VEL
LIN {X 0,Y 157.401,Z 604.882,A -85,B 0,C 180,E1 -23559.667,E2 -23559.667} C_VEL
LIN {X 0,Y 157.485,Z 604.87,A -85,B 0,C 180,E1 -23564.468,E2 -23564.468} C_VEL
LIN {X 0,Y 157.779,Z 604.834,A -85,B 0,C 180,E1 -23569.736,E2 -23569.736} C_VEL
LIN {X 0,Y 157.83,Z 604.823,A -85,B 0,C 180,E1 -23572.322,E2 -23572.322} C_VEL
LIN {X 0,Y 158.263,Z 604.771,A -85,B 0,C 180,E1 -23579.999,E2 -23579.999} C_VEL
LIN {X 0,Y 157.814,Z 604.819,A -85,B 0,C 180,E1 -23587.677,E2 -23587.677} C_VEL
LIN {X 0,Y 157.688,Z 604.841,A -85,B 0,C 180,E1 -23591.319,E2 -23591.319} C_VEL
LIN {X 0,Y 157.466,Z 604.846,A -85,B 0,C 180,E1 -23595.532,E2 -23595.532} C_VEL
LIN {X 0,Y 157.375,Z 604.882,A -85,B 0,C 180,E1 -23600.931,E2 -23600.931} C_VEL
LIN {X 0,Y 157.319,Z 604.867,A -85,B 0,C 180,E1 -23606.683,E2 -23606.683} C_VEL
LIN {X 0,Y 157.285,Z 604.893,A -85,B 0,C 180,E1 -23612.424,E2 -23612.424} C_VEL
LIN {X 0,Y 157.271,Z 604.896,A -85,B 0,C 180,E1 -23616.447,E2 -23616.447} C_VEL
LIN {X 0,Y 157.213,Z 604.898,A -85,B 0,C 180,E1 -23622.108,E2 -23622.108} C_VEL
LIN {X 0,Y 157.217,Z 604.898,A -85,B 0,C 180,E1 -23627.889,E2 -23627.889} C_VEL
LIN {X 0,Y 157.285,Z 604.885,A -85,B 0,C 180,E1 -23633.541,E2 -23633.541} C_VEL
LIN {X 0,Y 157.295,Z 604.882,A -85,B 0,C 180,E1 -23638.093,E2 -23638.093} C_VEL
LIN {X 0,Y 157.322,Z 604.881,A -85,B 0,C 180,E1 -23643.464,E2 -23643.464} C_VEL
LIN {X 0,Y 157.364,Z 604.884,A -85,B 0,C 180,E1 -23645.729,E2 -23645.729} C_VEL
LIN {X 0,Y 158.469,Z 607.901,A -85,B 0,C 180,E1 -23646.392,E2 -23646.392} C_VEL
LIN {X 0,Y 162.355,Z 616.059,A -85,B 0,C 180,E1 -23648.558,E2 -23648.558} C_VEL
LIN {X 0,Y 165.737,Z 624.746,A -85,B 0,C 180,E1 -23650.891,E2 -23650.891} C_VEL
LIN {X 0,Y 168.571,Z 634.066,A -85,B 0,C 180,E1 -23653.514,E2 -23653.514} C_VEL
LIN {X 0,Y 170.37,Z 642.2,A -85,B 0,C 180,E1 -23655.973,E2 -23655.973} C_VEL
LIN {X 0,Y 168.004,Z 651.794,A -85,B 0,C 180,E1 -23658.537,E2 -23658.537} C_VEL
LIN {X 0,Y 165.692,Z 660.546,A -85,B 0,C 180,E1 -23661.46,E2 -23661.46} C_VEL
LIN {X 0,Y 163.356,Z 669.085,A -85,B 0,C 180,E1 -23665.062,E2 -23665.062} C_VEL
LIN {X 0,Y 161.447,Z 675.757,A -85,B 0,C 180,E1 -23668.626,E2 -23668.626} C_VEL
LIN {X 0,Y 159.803,Z 681.508,A -85,B 0,C 180,E1 -23672.518,E2 -23672.518} C_VEL
LIN {X 0,Y 158.753,Z 685.874,A -85,B 0,C 180,E1 -23676.352,E2 -23676.352} C_VEL
LIN {X 0,Y 158.255,Z 689.172,A -85,B 0,C 180,E1 -23680.23,E2 -23680.23} C_VEL
LIN {X 0,Y 158.19,Z 690.84,A -85,B 0,C 180,E1 -23682.832,E2 -23682.832} C_VEL
LIN {X 0,Y 158.379,Z 692.077,A -85,B 0,C 180,E1 -23685.439,E2 -23685.439} C_VEL
LIN {X 0,Y 159.478,Z 693.298,A -85,B 0,C 180,E1 -23690.641,E2 -23690.641} C_VEL
LIN {X 0,Y 160.434,Z 693.32,A -85,B 0,C 180,E1 -23693.217,E2 -23693.217} C_VEL
LIN {X 0,Y 161.59,Z 692.903,A -85,B 0,C 180,E1 -23695.778,E2 -23695.778} C_VEL
LIN {X 0,Y 163.029,Z 692.069,A -85,B 0,C 180,E1 -23698.304,E2 -23698.304} C_VEL
LIN {X 0,Y 165.555,Z 690.114,A -85,B 0,C 180,E1 -23701.897,E2 -23701.897} C_VEL
LIN {X 0,Y 168.815,Z 686.955,A -85,B 0,C 180,E1 -23705.647,E2 -23705.647} C_VEL
LIN {X 0,Y 172.785,Z 682.423,A -85,B 0,C 180,E1 -23709.394,E2 -23709.394} C_VEL
LIN {X 0,Y 176.739,Z 677.281,A -85,B 0,C 180,E1 -23712.529,E2 -23712.529} C_VEL
LIN {X 0,Y 177.733,Z 675.836,A -85,B 0,C 180,E1 -23713.288,E2 -23713.288} C_VEL
LIN {X 0,Y 176.699,Z 675.007,A -85,B 0,C 180,E1 -23714.282,E2 -23714.282} C_VEL
LIN {X 0,Y 165.565,Z 673.729,A -85,B 0,C 180,E1 -23719.821,E2 -23719.821} C_VEL
LIN {X 0,Y 163.898,Z 673.065,A -85,B 0,C 180,E1 -23721.087,E2 -23721.087} C_VEL
LIN {X 0,Y 163.755,Z 672.818,A -85,B 0,C 180,E1 -23721.341,E2 -23721.341} C_VEL
LIN {X 0,Y 163.482,Z 677.517,A -85,B 0,C 180,E1 -23722.224,E2 -23722.224} C_VEL
LIN {X 0,Y 161.492,Z 689.633,A -85,B 0,C 180,E1 -23724.788,E2 -23724.788} C_VEL
LIN {X 0,Y 159.762,Z 700.137,A -85,B 0,C 180,E1 -23727.572,E2 -23727.572} C_VEL
LIN {X 0,Y 158.057,Z 709.817,A -85,B 0,C 180,E1 -23730.719,E2 -23730.719} C_VEL
LIN {X 0,Y 156.601,Z 719.83,A -85,B 0,C 180,E1 -23734.765,E2 -23734.765} C_VEL
LIN {X 0,Y 155.609,Z 727.923,A -85,B 0,C 180,E1 -23738.82,E2 -23738.82} C_VEL
LIN {X 0,Y 154.974,Z 734.755,A -85,B 0,C 180,E1 -23743.124,E2 -23743.124} C_VEL
LIN {X 0,Y 154.792,Z 739.504,A -85,B 0,C 180,E1 -23746.88,E2 -23746.88} C_VEL
LIN {X 0,Y 155.407,Z 744.697,A -85,B 0,C 180,E1 -23752.204,E2 -23752.204} C_VEL
LIN {X 0,Y 156.11,Z 746.66,A -85,B 0,C 180,E1 -23754.835,E2 -23754.835} C_VEL
LIN {X 0,Y 158.141,Z 749.375,A -85,B 0,C 180,E1 -23760.001,E2 -23760.001} C_VEL
LIN {X 0,Y 161.538,Z 750.705,A -85,B 0,C 180,E1 -23764.993,E2 -23764.993} C_VEL
LIN {X 0,Y 166.063,Z 750.59,A -85,B 0,C 180,E1 -23769.747,E2 -23769.747} C_VEL
LIN {X 0,Y 171.83,Z 749.076,A -85,B 0,C 180,E1 -23774.207,E2 -23774.207} C_VEL
LIN {X 0,Y 178.731,Z 746.184,A -85,B 0,C 180,E1 -23778.336,E2 -23778.336} C_VEL
LIN {X 0,Y 186.669,Z 741.693,A -85,B 0,C 180,E1 -23782.118,E2 -23782.118} C_VEL
LIN {X 0,Y 193.621,Z 737.016,A -85,B 0,C 180,E1 -23784.851,E2 -23784.851} C_VEL
LIN {X 0,Y 201.506,Z 730.805,A -85,B 0,C 180,E1 -23787.525,E2 -23787.525} C_VEL
LIN {X 0,Y 210.346,Z 722.72,A -85,B 0,C 180,E1 -23790.079,E2 -23790.079} C_VEL
LIN {X 0,Y 213.862,Z 718.497,A -85,B 0,C 180,E1 -23792.544,E2 -23792.544} C_VEL
LIN {X 0,Y 215.269,Z 716.777,A -85,B 0,C 180,E1 -23793.712,E2 -23793.712} C_VEL
LIN {X 0,Y 216.422,Z 715.352,A -85,B 0,C 180,E1 -23795.77,E2 -23795.77} C_VEL
LIN {X 0,Y 217.116,Z 714.858,A -85,B 0,C 180,E1 -23797.955,E2 -23797.955} C_VEL
LIN {X 0,Y 217.382,Z 714.994,A -85,B 0,C 180,E1 -23799.115,E2 -23799.115} C_VEL
LIN {X 0,Y 217.095,Z 715.685,A -85,B 0,C 180,E1 -23799.965,E2 -23799.965} C_VEL
LIN {X 0,Y 213.133,Z 721.043,A -85,B 0,C 180,E1 -23802.146,E2 -23802.146} C_VEL
LIN {X 0,Y 209.45,Z 725.671,A -85,B 0,C 180,E1 -23803.831,E2 -23803.831} C_VEL
LIN {X 0,Y 205.003,Z 730.654,A -85,B 0,C 180,E1 -23805.352,E2 -23805.352} C_VEL
LIN {X 0,Y 195.675,Z 739.743,A -85,B 0,C 180,E1 -23808.362,E2 -23808.362} C_VEL
LIN {X 0,Y 189.047,Z 745.53,A -85,B 0,C 180,E1 -23810.806,E2 -23810.806} C_VEL
LIN {X 0,Y 180.485,Z 751.896,A -85,B 0,C 180,E1 -23814.264,E2 -23814.264} C_VEL
LIN {X 0,Y 173.184,Z 756.787,A -85,B 0,C 180,E1 -23818.162,E2 -23818.162} C_VEL
LIN {X 0,Y 166.85,Z 760.345,A -85,B 0,C 180,E1 -23822.4,E2 -23822.4} C_VEL
LIN {X 0,Y 161.973,Z 762.571,A -85,B 0,C 180,E1 -23827.017,E2 -23827.017} C_VEL
